LIN {X 0,Y 253.326,Z 243.578,A -85,B 0,C 180,E1 -18994.775,E2 -18994.775} C_VEL
LIN {X 0,Y 254.902,Z 232.784,A -85,B 0,C 180,E1 -18996.591,E2 -18996.591} C_VEL
LIN {X 0,Y 256.298,Z 221.635,A -85,B 0,C 180,E1 -18998.079,E2 -18998.079} C_VEL
LIN {X 0,Y 257.475,Z 209.502,A -85,B 0,C 180,E1 -18999.328,E2 -18999.328} C_VEL
LIN {X 0,Y 258.563,Z 195.963,A -85,B 0,C 180,E1 -19000.325,E2 -19000.325} C_VEL
LIN {X 0,Y 259.185,Z 183.358,A -85,B 0,C 180,E1 -19000.942,E2 -19000.942} C_VEL
LIN {X 0,Y 261.265,Z 111.221,A -85,B 0,C 180,E1 -19002.915,E2 -19002.915} C_VEL
LIN {X 0,Y 257.099,Z 99.785,A -85,B 0,C 180,E1 -19003.638,E2 -19003.638} C_VEL
LIN {X 0,Y 249.447,Z 82.487,A -85,B 0,C 180,E1 -19004.922,E2 -19004.922} C_VEL
LIN {X 0,Y 249.249,Z 81.443,A -85,B 0,C 180,E1 -19005.015,E2 -19005.015} C_VEL
LIN {X 0,Y 249.144,Z 81.454,A -85,B 0,C 180,E1 -19008.078,E2 -19008.078} C_VEL
LIN {X 0,Y 249.089,Z 81.456,A -85,B 0,C 180,E1 -19011.519,E2 -19011.519} C_VEL
LIN {X 0,Y 249.122,Z 81.453,A -85,B 0,C 180,E1 -19015.476,E2 -19015.476} C_VEL
LIN {X 0,Y 249.078,Z 81.456,A -85,B 0,C 180,E1 -19018.989,E2 -19018.989} C_VEL
LIN {X 0,Y 249.041,Z 81.457,A -85,B 0,C 180,E1 -19022.425,E2 -19022.425} C_VEL
LIN {X 0,Y 249.074,Z 81.457,A -85,B 0,C 180,E1 -19026.339,E2 -19026.339} C_VEL
LIN {X 0,Y 249.036,Z 81.46,A -85,B 0,C 180,E1 -19030.473,E2 -19030.473} C_VEL
LIN {X 0,Y 249.014,Z 81.463,A -85,B 0,C 180,E1 -19034.877,E2 -19034.877} C_VEL
LIN {X 0,Y 249.022,Z 81.466,A -85,B 0,C 180,E1 -19037.363,E2 -19037.363} C_VEL
LIN {X 0,Y 249.047,Z 81.448,A -85,B 0,C 180,E1 -19042.2,E2 -19042.2} C_VEL
LIN {X 0,Y 249.047,Z 81.441,A -85,B 0,C 180,E1 -19045.639,E2 -19045.639} C_VEL
LIN {X 0,Y 249.051,Z 81.459,A -85,B 0,C 180,E1 -19049.472,E2 -19049.472} C_VEL
LIN {X 0,Y 249.075,Z 81.456,A -85,B 0,C 180,E1 -19053.162,E2 -19053.162} C_VEL
LIN {X 0,Y 249.083,Z 81.454,A -85,B 0,C 180,E1 -19056.732,E2 -19056.732} C_VEL
LIN {X 0,Y 249.115,Z 81.455,A -85,B 0,C 180,E1 -19060.211,E2 -19060.211} C_VEL
LIN {X 0,Y 249.245,Z 81.429,A -85,B 0,C 180,E1 -19063.622,E2 -19063.622} C_VEL
LIN {X 0,Y 249.248,Z 81.436,A -85,B 0,C 180,E1 -19068.616,E2 -19068.616} C_VEL
LIN {X 0,Y 249.458,Z 81.405,A -85,B 0,C 180,E1 -19071.902,E2 -19071.902} C_VEL
LIN {X 0,Y 249.298,Z 81.429,A -85,B 0,C 180,E1 -19075.148,E2 -19075.148} C_VEL
LIN {X 0,Y 249.678,Z 81.379,A -85,B 0,C 180,E1 -19078.387,E2 -19078.387} C_VEL
LIN {X 0,Y 249.678,Z 81.379,A -85,B 0,C 180,E1 -19081.613,E2 -19081.613} C_VEL
LIN {X 0,Y 249.449,Z 81.408,A -85,B 0,C 180,E1 -19086.47,E2 -19086.47} C_VEL
LIN {X 0,Y 249.345,Z 81.425,A -85,B 0,C 180,E1 -19089.736,E2 -19089.736} C_VEL
LIN {X 0,Y 249.242,Z 81.438,A -85,B 0,C 180,E1 -19091.224,E2 -19091.224} C_VEL
LIN {X 0,Y 248.557,Z 81.529,A -85,B 0,C 180,E1 -19092.572,E2 -19092.572} C_VEL
LIN {X 0,Y 245.654,Z 81.885,A -85,B 0,C 180,E1 -19094.769,E2 -19094.769} C_VEL
LIN {X 0,Y 243.198,Z 82.185,A -85,B 0,C 180,E1 -19096.558,E2 -19096.558} C_VEL
LIN {X 0,Y 242.153,Z 82.319,A -85,B 0,C 180,E1 -19097.948,E2 -19097.948} C_VEL
LIN {X 0,Y 242.072,Z 82.328,A -85,B 0,C 180,E1 -19098.419,E2 -19098.419} C_VEL
LIN {X 0,Y 242.009,Z 82.336,A -85,B 0,C 180,E1 -19102.18,E2 -19102.18} C_VEL
LIN {X 0,Y 242.069,Z 82.328,A -85,B 0,C 180,E1 -19105.838,E2 -19105.838} C_VEL
LIN {X 0,Y 242.032,Z 82.329,A -85,B 0,C 180,E1 -19109.58,E2 -19109.58} C_VEL
LIN {X 0,Y 241.982,Z 82.341,A -85,B 0,C 180,E1 -19113.492,E2 -19113.492} C_VEL
LIN {X 0,Y 241.991,Z 82.34,A -85,B 0,C 180,E1 -19117.581,E2 -19117.581} C_VEL
LIN {X 0,Y 241.939,Z 82.348,A -85,B 0,C 180,E1 -19121.922,E2 -19121.922} C_VEL
LIN {X 0,Y 241.936,Z 82.349,A -85,B 0,C 180,E1 -19126.571,E2 -19126.571} C_VEL
LIN {X 0,Y 241.974,Z 82.346,A -85,B 0,C 180,E1 -19130.284,E2 -19130.284} C_VEL
LIN {X 0,Y 242.047,Z 82.472,A -85,B 0,C 180,E1 -19133.859,E2 -19133.859} C_VEL
LIN {X 0,Y 244.076,Z 91.796,A -85,B 0,C 180,E1 -19137.323,E2 -19137.323} C_VEL
LIN {X 0,Y 245.923,Z 100.895,A -85,B 0,C 180,E1 -19140.533,E2 -19140.533} C_VEL
LIN {X 0,Y 248.2,Z 107.794,A -85,B 0,C 180,E1 -19140.981,E2 -19140.981} C_VEL
LIN {X 0,Y 253.338,Z 152.439,A -85,B 0,C 180,E1 -19142.841,E2 -19142.841} C_VEL
LIN {X 0,Y 253.472,Z 159.178,A -85,B 0,C 180,E1 -19143.057,E2 -19143.057} C_VEL
LIN {X 0,Y 251.997,Z 209.848,A -85,B 0,C 180,E1 -19144.498,E2 -19144.498} C_VEL
LIN {X 0,Y 251.014,Z 223.134,A -85,B 0,C 180,E1 -19145.166,E2 -19145.166} C_VEL
LIN {X 0,Y 249.809,Z 235.947,A -85,B 0,C 180,E1 -19146.145,E2 -19146.145} C_VEL
LIN {X 0,Y 248.331,Z 247.285,A -85,B 0,C 180,E1 -19147.318,E2 -19147.318} C_VEL
LIN {X 0,Y 246.817,Z 257.715,A -85,B 0,C 180,E1 -19148.712,E2 -19148.712} C_VEL
LIN {X 0,Y 245.466,Z 266.328,A -85,B 0,C 180,E1 -19150.123,E2 -19150.123} C_VEL
LIN {X 0,Y 243.8,Z 276.342,A -85,B 0,C 180,E1 -19152.152,E2 -19152.152} C_VEL
LIN {X 0,Y 242.667,Z 283.898,A -85,B 0,C 180,E1 -19154.029,E2 -19154.029} C_VEL
LIN {X 0,Y 241.426,Z 292.111,A -85,B 0,C 180,E1 -19156.533,E2 -19156.533} C_VEL
LIN {X 0,Y 240.582,Z 298.702,A -85,B 0,C 180,E1 -19159.054,E2 -19159.054} C_VEL
LIN {X 0,Y 240.155,Z 303.924,A -85,B 0,C 180,E1 -19161.586,E2 -19161.586} C_VEL
LIN {X 0,Y 240.024,Z 308.554,A -85,B 0,C 180,E1 -19164.581,E2 -19164.581} C_VEL
LIN {X 0,Y 240.045,Z 310.915,A -85,B 0,C 180,E1 -19166.642,E2 -19166.642} C_VEL
LIN {X 0,Y 240.096,Z 312.31,A -85,B 0,C 180,E1 -19168.322,E2 -19168.322} C_VEL
LIN {X 0,Y 240.155,Z 313.289,A -85,B 0,C 180,E1 -19169.999,E2 -19169.999} C_VEL
LIN {X 0,Y 240.034,Z 313.858,A -85,B 0,C 180,E1 -19171.677,E2 -19171.677} C_VEL
LIN {X 0,Y 239.963,Z 314.034,A -85,B 0,C 180,E1 -19173.357,E2 -19173.357} C_VEL
LIN {X 0,Y 239.911,Z 313.751,A -85,B 0,C 180,E1 -19175.126,E2 -19175.126} C_VEL
LIN {X 0,Y 240.132,Z 312.096,A -85,B 0,C 180,E1 -19178.414,E2 -19178.414} C_VEL
LIN {X 0,Y 240.485,Z 310.677,A -85,B 0,C 180,E1 -19180.098,E2 -19180.098} C_VEL
LIN {X 0,Y 241.291,Z 307.724,A -85,B 0,C 180,E1 -19182.617,E2 -19182.617} C_VEL
LIN {X 0,Y 242.716,Z 303.775,A -85,B 0,C 180,E1 -19185.105,E2 -19185.105} C_VEL
LIN {X 0,Y 244.543,Z 298.725,A -85,B 0,C 180,E1 -19187.563,E2 -19187.563} C_VEL
LIN {X 0,Y 246.699,Z 292.425,A -85,B 0,C 180,E1 -19189.989,E2 -19189.989} C_VEL
LIN {X 0,Y 249.454,Z 284.587,A -85,B 0,C 180,E1 -19192.354,E2 -19192.354} C_VEL
LIN {X 0,Y 252.756,Z 274.849,A -85,B 0,C 180,E1 -19194.65,E2 -19194.65} C_VEL
LIN {X 0,Y 255.766,Z 264.803,A -85,B 0,C 180,E1 -19196.52,E2 -19196.52} C_VEL
LIN {X 0,Y 258.886,Z 253.45,A -85,B 0,C 180,E1 -19198.143,E2 -19198.143} C_VEL
LIN {X 0,Y 261.47,Z 242.35,A -85,B 0,C 180,E1 -19199.375,E2 -19199.375} C_VEL
LIN {X 0,Y 263.807,Z 230.005,A -85,B 0,C 180,E1 -19200.409,E2 -19200.409} C_VEL
LIN {X 0,Y 265.654,Z 216.896,A -85,B 0,C 180,E1 -19201.166,E2 -19201.166} C_VEL
LIN {X 0,Y 266.696,Z 204.407,A -85,B 0,C 180,E1 -19201.639,E2 -19201.639} C_VEL
LIN {X 0,Y 268.491,Z 159.915,A -85,B 0,C 180,E1 -19202.843,E2 -19202.843} C_VEL
LIN {X 0,Y 265.485,Z 139.44,A -85,B 0,C 180,E1 -19204.05,E2 -19204.05} C_VEL
LIN {X 0,Y 264.082,Z 132.709,A -85,B 0,C 180,E1 -19204.533,E2 -19204.533} C_VEL
LIN {X 0,Y 256.737,Z 117.087,A -85,B 0,C 180,E1 -19206.475,E2 -19206.475} C_VEL
LIN {X 0,Y 250.909,Z 106.205,A -85,B 0,C 180,E1 -19208.088,E2 -19208.088} C_VEL
LIN {X 0,Y 248.94,Z 102.739,A -85,B 0,C 180,E1 -19208.652,E2 -19208.652} C_VEL
LIN {X 0,Y 246.669,Z 98.329,A -85,B 0,C 180,E1 -19209.374,E2 -19209.374} C_VEL
LIN {X 0,Y 244.126,Z 89.558,A -85,B 0,C 180,E1 -19213.702,E2 -19213.702} C_VEL
LIN {X 0,Y 241.982,Z 82.339,A -85,B 0,C 180,E1 -19217.689,E2 -19217.689} C_VEL
LIN {X 0,Y 242.008,Z 82.331,A -85,B 0,C 180,E1 -19222.422,E2 -19222.422} C_VEL
LIN {X 0,Y 241.989,Z 82.336,A -85,B 0,C 180,E1 -19226.509,E2 -19226.509} C_VEL
LIN {X 0,Y 242.035,Z 82.333,A -85,B 0,C 180,E1 -19230.587,E2 -19230.587} C_VEL
LIN {X 0,Y 242.065,Z 82.324,A -85,B 0,C 180,E1 -19234.183,E2 -19234.183} C_VEL
LIN {X 0,Y 242.051,Z 82.322,A -85,B 0,C 180,E1 -19238.297,E2 -19238.297} C_VEL
LIN {X 0,Y 242.161,Z 82.311,A -85,B 0,C 180,E1 -19243.278,E2 -19243.278} C_VEL
LIN {X 0,Y 242.184,Z 82.306,A -85,B 0,C 180,E1 -19248.28,E2 -19248.28} C_VEL
LIN {X 0,Y 242.424,Z 82.274,A -85,B 0,C 180,E1 -19251.666,E2 -19251.666} C_VEL
LIN {X 0,Y 242.256,Z 82.309,A -85,B 0,C 180,E1 -19255.007,E2 -19255.007} C_VEL
LIN {X 0,Y 242.634,Z 82.248,A -85,B 0,C 180,E1 -19258.341,E2 -19258.341} C_VEL
LIN {X 0,Y 242.633,Z 82.252,A -85,B 0,C 180,E1 -19261.66,E2 -19261.66} C_VEL
LIN {X 0,Y 242.414,Z 82.282,A -85,B 0,C 180,E1 -19266.671,E2 -19266.671} C_VEL
LIN {X 0,Y 242.264,Z 82.307,A -85,B 0,C 180,E1 -19270.024,E2 -19270.024} C_VEL
LIN {X 0,Y 242.137,Z 82.324,A -85,B 0,C 180,E1 -19275.143,E2 -19275.143} C_VEL
LIN {X 0,Y 242.048,Z 82.327,A -85,B 0,C 180,E1 -19278.627,E2 -19278.627} C_VEL
LIN {X 0,Y 242.002,Z 82.329,A -85,B 0,C 180,E1 -19282.182,E2 -19282.182} C_VEL
LIN {X 0,Y 242.031,Z 82.327,A -85,B 0,C 180,E1 -19285.822,E2 -19285.822} C_VEL
LIN {X 0,Y 241.969,Z 82.337,A -85,B 0,C 180,E1 -19289.589,E2 -19289.589} C_VEL
LIN {X 0,Y 241.978,Z 82.342,A -85,B 0,C 180,E1 -19293.494,E2 -19293.494} C_VEL
LIN {X 0,Y 241.988,Z 82.338,A -85,B 0,C 180,E1 -19295.656,E2 -19295.656} C_VEL
LIN {X 0,Y 242.945,Z 85.113,A -85,B 0,C 180,E1 -19296.016,E2 -19296.016} C_VEL
LIN {X 0,Y 245.321,Z 87.875,A -85,B 0,C 180,E1 -19296.704,E2 -19296.704} C_VEL
LIN {X 0,Y 247.518,Z 91.21,A -85,B 0,C 180,E1 -19297.349,E2 -19297.349} C_VEL
LIN {X 0,Y 255.952,Z 103.808,A -85,B 0,C 180,E1 -19299.658,E2 -19299.658} C_VEL
LIN {X 0,Y 263.759,Z 117.045,A -85,B 0,C 180,E1 -19301.642,E2 -19301.642} C_VEL
LIN {X 0,Y 269.885,Z 129.938,A -85,B 0,C 180,E1 -19303.166,E2 -19303.166} C_VEL
LIN {X 0,Y 267.385,Z 185.069,A -85,B 0,C 180,E1 -19304.641,E2 -19304.641} C_VEL
LIN {X 0,Y 266.192,Z 198.279,A -85,B 0,C 180,E1 -19305.267,E2 -19305.267} C_VEL
LIN {X 0,Y 264.735,Z 210.283,A -85,B 0,C 180,E1 -19306.133,E2 -19306.133} C_VEL
LIN {X 0,Y 262.688,Z 221.975,A -85,B 0,C 180,E1 -19307.244,E2 -19307.244} C_VEL
LIN {X 0,Y 260.354,Z 232.814,A -85,B 0,C 180,E1 -19308.598,E2 -19308.598} C_VEL
LIN {X 0,Y 257.378,Z 244.089,A -85,B 0,C 180,E1 -19310.39,E2 -19310.39} C_VEL
LIN {X 0,Y 254.767,Z 252.802,A -85,B 0,C 180,E1 -19312.137,E2 -19312.137} C_VEL
LIN {X 0,Y 252.064,Z 260.954,A -85,B 0,C 180,E1 -19314.161,E2 -19314.161} C_VEL
LIN {X 0,Y 249.231,Z 268.801,A -85,B 0,C 180,E1 -19316.642,E2 -19316.642} C_VEL
LIN {X 0,Y 246.777,Z 275.025,A -85,B 0,C 180,E1 -19319.162,E2 -19319.162} C_VEL
LIN {X 0,Y 244.728,Z 279.883,A -85,B 0,C 180,E1 -19321.717,E2 -19321.717} C_VEL
LIN {X 0,Y 243.121,Z 283.537,A -85,B 0,C 180,E1 -19324.304,E2 -19324.304} C_VEL
LIN {X 0,Y 242.244,Z 285.369,A -85,B 0,C 180,E1 -19326.036,E2 -19326.036} C_VEL
LIN {X 0,Y 241.125,Z 287.353,A -85,B 0,C 180,E1 -19328.861,E2 -19328.861} C_VEL
LIN {X 0,Y 240.43,Z 288.166,A -85,B 0,C 180,E1 -19331.245,E2 -19331.245} C_VEL
LIN {X 0,Y 240.119,Z 288.226,A -85,B 0,C 180,E1 -19332.982,E2 -19332.982} C_VEL
LIN {X 0,Y 239.941,Z 287.748,A -85,B 0,C 180,E1 -19335.15,E2 -19335.15} C_VEL
LIN {X 0,Y 239.923,Z 285.974,A -85,B 0,C 180,E1 -19338.168,E2 -19338.168} C_VEL
LIN {X 0,Y 240.215,Z 283.416,A -85,B 0,C 180,E1 -19340.741,E2 -19340.741} C_VEL
LIN {X 0,Y 240.691,Z 279.845,A -85,B 0,C 180,E1 -19343.293,E2 -19343.293} C_VEL
LIN {X 0,Y 241.299,Z 275.174,A -85,B 0,C 180,E1 -19345.825,E2 -19345.825} C_VEL
LIN {X 0,Y 242.331,Z 268.136,A -85,B 0,C 180,E1 -19348.754,E2 -19348.754} C_VEL
LIN {X 0,Y 243.634,Z 260.515,A -85,B 0,C 180,E1 -19351.24,E2 -19351.24} C_VEL
LIN {X 0,Y 245.003,Z 252.706,A -85,B 0,C 180,E1 -19353.289,E2 -19353.289} C_VEL
LIN {X 0,Y 246.762,Z 242.095,A -85,B 0,C 180,E1 -19355.517,E2 -19355.517} C_VEL
LIN {X 0,Y 248.368,Z 231.465,A -85,B 0,C 180,E1 -19357.29,E2 -19357.29} C_VEL
LIN {X 0,Y 249.678,Z 220.807,A -85,B 0,C 180,E1 -19358.703,E2 -19358.703} C_VEL
LIN {X 0,Y 250.81,Z 209.345,A -85,B 0,C 180,E1 -19359.883,E2 -19359.883} C_VEL
LIN {X 0,Y 251.895,Z 196.367,A -85,B 0,C 180,E1 -19360.856,E2 -19360.856} C_VEL
LIN {X 0,Y 252.569,Z 183.311,A -85,B 0,C 180,E1 -19361.504,E2 -19361.504} C_VEL
LIN {X 0,Y 254.778,Z 112.933,A -85,B 0,C 180,E1 -19363.459,E2 -19363.459} C_VEL
LIN {X 0,Y 250.712,Z 101.974,A -85,B 0,C 180,E1 -19364.188,E2 -19364.188} C_VEL
LIN {X 0,Y 242.289,Z 82.759,A -85,B 0,C 180,E1 -19365.676,E2 -19365.676} C_VEL
LIN {X 0,Y 242.22,Z 82.318,A -85,B 0,C 180,E1 -19365.705,E2 -19365.705} C_VEL
LIN {X 0,Y 242.041,Z 82.337,A -85,B 0,C 180,E1 -19370.392,E2 -19370.392} C_VEL
LIN {X 0,Y 242.046,Z 82.334,A -85,B 0,C 180,E1 -19373.986,E2 -19373.986} C_VEL
LIN {X 0,Y 242.005,Z 82.332,A -85,B 0,C 180,E1 -19377.688,E2 -19377.688} C_VEL
LIN {X 0,Y 241.98,Z 82.343,A -85,B 0,C 180,E1 -19381.52,E2 -19381.52} C_VEL
LIN {X 0,Y 242.033,Z 82.331,A -85,B 0,C 180,E1 -19385.604,E2 -19385.604} C_VEL
LIN {X 0,Y 241.98,Z 82.34,A -85,B 0,C 180,E1 -19389.715,E2 -19389.715} C_VEL
LIN {X 0,Y 241.945,Z 82.342,A -85,B 0,C 180,E1 -19394.199,E2 -19394.199} C_VEL
LIN {X 0,Y 241.943,Z 82.345,A -85,B 0,C 180,E1 -19398.078,E2 -19398.078} C_VEL
LIN {X 0,Y 241.99,Z 82.325,A -85,B 0,C 180,E1 -19402.417,E2 -19402.417} C_VEL
LIN {X 0,Y 241.984,Z 82.323,A -85,B 0,C 180,E1 -19406.507,E2 -19406.507} C_VEL
LIN {X 0,Y 242.017,Z 82.337,A -85,B 0,C 180,E1 -19410.597,E2 -19410.597} C_VEL
LIN {X 0,Y 242.071,Z 82.328,A -85,B 0,C 180,E1 -19414.183,E2 -19414.183} C_VEL
LIN {X 0,Y 242.057,Z 82.332,A -85,B 0,C 180,E1 -19418.297,E2 -19418.297} C_VEL
LIN {X 0,Y 242.167,Z 82.31,A -85,B 0,C 180,E1 -19423.278,E2 -19423.278} C_VEL
LIN {X 0,Y 242.184,Z 82.318,A -85,B 0,C 180,E1 -19428.279,E2 -19428.279} C_VEL
LIN {X 0,Y 242.404,Z 82.283,A -85,B 0,C 180,E1 -19431.664,E2 -19431.664} C_VEL
LIN {X 0,Y 242.259,Z 82.305,A -85,B 0,C 180,E1 -19435.007,E2 -19435.007} C_VEL
LIN {X 0,Y 242.638,Z 82.256,A -85,B 0,C 180,E1 -19438.34,E2 -19438.34} C_VEL
LIN {X 0,Y 242.638,Z 82.256,A -85,B 0,C 180,E1 -19441.659,E2 -19441.659} C_VEL
LIN {X 0,Y 242.419,Z 82.283,A -85,B 0,C 180,E1 -19446.659,E2 -19446.659} C_VEL
LIN {X 0,Y 242.269,Z 82.305,A -85,B 0,C 180,E1 -19450.023,E2 -19450.023} C_VEL
LIN {X 0,Y 242.169,Z 82.314,A -85,B 0,C 180,E1 -19455.14,E2 -19455.14} C_VEL
LIN {X 0,Y 242.072,Z 82.328,A -85,B 0,C 180,E1 -19458.419,E2 -19458.419} C_VEL
LIN {X 0,Y 241.403,Z 82.42,A -85,B 0,C 180,E1 -19459.807,E2 -19459.807} C_VEL
LIN {X 0,Y 238.508,Z 82.78,A -85,B 0,C 180,E1 -19462.069,E2 -19462.069} C_VEL
LIN {X 0,Y 236.063,Z 83.078,A -85,B 0,C 180,E1 -19463.913,E2 -19463.913} C_VEL
LIN {X 0,Y 235.044,Z 83.204,A -85,B 0,C 180,E1 -19465.346,E2 -19465.346} C_VEL
LIN {X 0,Y 234.978,Z 83.211,A -85,B 0,C 180,E1 -19465.831,E2 -19465.831} C_VEL
LIN {X 0,Y 234.934,Z 83.213,A -85,B 0,C 180,E1 -19470.567,E2 -19470.567} C_VEL
LIN {X 0,Y 234.932,Z 83.221,A -85,B 0,C 180,E1 -19474.637,E2 -19474.637} C_VEL
LIN {X 0,Y 234.943,Z 83.217,A -85,B 0,C 180,E1 -19478.944,E2 -19478.944} C_VEL
LIN {X 0,Y 234.889,Z 83.222,A -85,B 0,C 180,E1 -19483.485,E2 -19483.485} C_VEL
LIN {X 0,Y 234.889,Z 83.227,A -85,B 0,C 180,E1 -19486.514,E2 -19486.514} C_VEL
LIN {X 0,Y 234.956,Z 83.22,A -85,B 0,C 180,E1 -19491.086,E2 -19491.086} C_VEL
LIN {X 0,Y 234.994,Z 83.241,A -85,B 0,C 180,E1 -19493.262,E2 -19493.262} C_VEL
LIN {X 0,Y 237.003,Z 92.535,A -85,B 0,C 180,E1 -19496.84,E2 -19496.84} C_VEL
LIN {X 0,Y 238.655,Z 100.654,A -85,B 0,C 180,E1 -19499.751,E2 -19499.751} C_VEL
LIN {X 0,Y 241.824,Z 109.835,A -85,B 0,C 180,E1 -19500.391,E2 -19500.391} C_VEL
LIN {X 0,Y 246.655,Z 152.06,A -85,B 0,C 180,E1 -19502.213,E2 -19502.213} C_VEL
LIN {X 0,Y 246.901,Z 159.165,A -85,B 0,C 180,E1 -19502.458,E2 -19502.458} C_VEL
LIN {X 0,Y 245.349,Z 209.737,A -85,B 0,C 180,E1 -19503.933,E2 -19503.933} C_VEL
LIN {X 0,Y 244.291,Z 223.619,A -85,B 0,C 180,E1 -19504.663,E2 -19504.663} C_VEL
LIN {X 0,Y 243.041,Z 236.191,A -85,B 0,C 180,E1 -19505.665,E2 -19505.665} C_VEL
LIN {X 0,Y 241.514,Z 247.358,A -85,B 0,C 180,E1 -19506.868,E2 -19506.868} C_VEL
LIN {X 0,Y 239.954,Z 257.708,A -85,B 0,C 180,E1 -19508.298,E2 -19508.298} C_VEL
LIN {X 0,Y 238.562,Z 266.26,A -85,B 0,C 180,E1 -19509.747,E2 -19509.747} C_VEL
LIN {X 0,Y 236.806,Z 276.349,A -85,B 0,C 180,E1 -19511.861,E2 -19511.861} C_VEL
LIN {X 0,Y 235.515,Z 284.49,A -85,B 0,C 180,E1 -19513.976,E2 -19513.976} C_VEL
LIN {X 0,Y 234.268,Z 292.53,A -85,B 0,C 180,E1 -19516.555,E2 -19516.555} C_VEL
LIN {X 0,Y 233.555,Z 297.962,A -85,B 0,C 180,E1 -19518.72,E2 -19518.72} C_VEL
LIN {X 0,Y 233.095,Z 303.268,A -85,B 0,C 180,E1 -19521.329,E2 -19521.329} C_VEL
LIN {X 0,Y 232.935,Z 307.488,A -85,B 0,C 180,E1 -19524.025,E2 -19524.025} C_VEL
LIN {X 0,Y 232.957,Z 310.378,A -85,B 0,C 180,E1 -19526.54,E2 -19526.54} C_VEL
LIN {X 0,Y 233.021,Z 311.828,A -85,B 0,C 180,E1 -19528.271,E2 -19528.271} C_VEL
LIN {X 0,Y 233.075,Z 312.834,A -85,B 0,C 180,E1 -19529.999,E2 -19529.999} C_VEL
LIN {X 0,Y 232.959,Z 313.431,A -85,B 0,C 180,E1 -19531.728,E2 -19531.728} C_VEL
LIN {X 0,Y 232.878,Z 313.637,A -85,B 0,C 180,E1 -19533.46,E2 -19533.46} C_VEL
LIN {X 0,Y 232.839,Z 313.434,A -85,B 0,C 180,E1 -19535.195,E2 -19535.195} C_VEL
LIN {X 0,Y 233.08,Z 311.809,A -85,B 0,C 180,E1 -19538.671,E2 -19538.671} C_VEL
LIN {X 0,Y 233.466,Z 310.42,A -85,B 0,C 180,E1 -19540.405,E2 -19540.405} C_VEL
LIN {X 0,Y 234.33,Z 307.529,A -85,B 0,C 180,E1 -19542.999,E2 -19542.999} C_VEL
LIN {X 0,Y 235.854,Z 303.646,A -85,B 0,C 180,E1 -19545.555,E2 -19545.555} C_VEL
LIN {X 0,Y 237.77,Z 298.666,A -85,B 0,C 180,E1 -19548.08,E2 -19548.08} C_VEL
LIN {X 0,Y 240.035,Z 292.442,A -85,B 0,C 180,E1 -19550.569,E2 -19550.569} C_VEL
LIN {X 0,Y 242.902,Z 284.737,A -85,B 0,C 180,E1 -19552.991,E2 -19552.991} C_VEL
LIN {X 0,Y 246.342,Z 275.105,A -85,B 0,C 180,E1 -19555.336,E2 -19555.336} C_VEL
LIN {X 0,Y 249.46,Z 265.208,A -85,B 0,C 180,E1 -19557.245,E2 -19557.245} C_VEL
LIN {X 0,Y 252.69,Z 254.091,A -85,B 0,C 180,E1 -19558.897,E2 -19558.897} C_VEL
LIN {X 0,Y 255.343,Z 243.237,A -85,B 0,C 180,E1 -19560.152,E2 -19560.152} C_VEL
LIN {X 0,Y 257.75,Z 231.286,A -85,B 0,C 180,E1 -19561.202,E2 -19561.202} C_VEL
LIN {X 0,Y 259.732,Z 218.262,A -85,B 0,C 180,E1 -19562.017,E2 -19562.017} C_VEL
LIN {X 0,Y 260.945,Z 205.409,A -85,B 0,C 180,E1 -19562.534,E2 -19562.534} C_VEL
LIN {X 0,Y 262.874,Z 160.81,A -85,B 0,C 180,E1 -19563.766,E2 -19563.766} C_VEL
LIN {X 0,Y 259.723,Z 139.333,A -85,B 0,C 180,E1 -19565.093,E2 -19565.093} C_VEL
LIN {X 0,Y 258.858,Z 135.778,A -85,B 0,C 180,E1 -19565.382,E2 -19565.382} C_VEL
LIN {X 0,Y 252.112,Z 121.264,A -85,B 0,C 180,E1 -19567.252,E2 -19567.252} C_VEL
LIN {X 0,Y 245.295,Z 108.243,A -85,B 0,C 180,E1 -19569.251,E2 -19569.251} C_VEL
LIN {X 0,Y 241.807,Z 102.388,A -85,B 0,C 180,E1 -19570.314,E2 -19570.314} C_VEL
LIN {X 0,Y 239.248,Z 97.728,A -85,B 0,C 180,E1 -19571.193,E2 -19571.193} C_VEL
LIN {X 0,Y 236.609,Z 88.756,A -85,B 0,C 180,E1 -19575.958,E2 -19575.958} C_VEL
LIN {X 0,Y 234.924,Z 83.215,A -85,B 0,C 180,E1 -19579.267,E2 -19579.267} C_VEL
LIN {X 0,Y 234.955,Z 83.218,A -85,B 0,C 180,E1 -19583.863,E2 -19583.863} C_VEL
LIN {X 0,Y 234.958,Z 83.219,A -85,B 0,C 180,E1 -19587.425,E2 -19587.425} C_VEL
LIN {X 0,Y 234.95,Z 83.219,A -85,B 0,C 180,E1 -19591.406,E2 -19591.406} C_VEL
LIN {X 0,Y 234.986,Z 83.215,A -85,B 0,C 180,E1 -19595.247,E2 -19595.247} C_VEL
LIN {X 0,Y 235.01,Z 83.205,A -85,B 0,C 180,E1 -19598.97,E2 -19598.97} C_VEL
LIN {X 0,Y 235.094,Z 83.189,A -85,B 0,C 180,E1 -19603.059,E2 -19603.059} C_VEL
LIN {X 0,Y 235.116,Z 83.183,A -85,B 0,C 180,E1 -19607.922,E2 -19607.922} C_VEL
LIN {X 0,Y 235.374,Z 83.154,A -85,B 0,C 180,E1 -19611.414,E2 -19611.414} C_VEL
LIN {X 0,Y 235.4,Z 83.148,A -85,B 0,C 180,E1 -19613.142,E2 -19613.142} C_VEL
LIN {X 0,Y 235.593,Z 83.124,A -85,B 0,C 180,E1 -19618.291,E2 -19618.291} C_VEL
LIN {X 0,Y 235.593,Z 83.128,A -85,B 0,C 180,E1 -19621.71,E2 -19621.71} C_VEL
LIN {X 0,Y 235.365,Z 83.157,A -85,B 0,C 180,E1 -19626.86,E2 -19626.86} C_VEL
LIN {X 0,Y 235.21,Z 83.187,A -85,B 0,C 180,E1 -19630.328,E2 -19630.328} C_VEL
LIN {X 0,Y 235.084,Z 83.202,A -85,B 0,C 180,E1 -19635.609,E2 -19635.609} C_VEL
LIN {X 0,Y 234.989,Z 83.211,A -85,B 0,C 180,E1 -19639.208,E2 -19639.208} C_VEL
LIN {X 0,Y 234.948,Z 83.212,A -85,B 0,C 180,E1 -19642.885,E2 -19642.885} C_VEL
LIN {X 0,Y 234.945,Z 83.213,A -85,B 0,C 180,E1 -19646.661,E2 -19646.661} C_VEL
LIN {X 0,Y 234.898,Z 83.224,A -85,B 0,C 180,E1 -19650.573,E2 -19650.573} C_VEL
LIN {X 0,Y 234.923,Z 83.224,A -85,B 0,C 180,E1 -19653.849,E2 -19653.849} C_VEL
LIN {X 0,Y 235.728,Z 85.726,A -85,B 0,C 180,E1 -19654.189,E2 -19654.189} C_VEL
LIN {X 0,Y 237.702,Z 88.027,A -85,B 0,C 180,E1 -19654.816,E2 -19654.816} C_VEL
LIN {X 0,Y 238.457,Z 88.997,A -85,B 0,C 180,E1 -19655.055,E2 -19655.055} C_VEL
LIN {X 0,Y 240.8,Z 92.379,A -85,B 0,C 180,E1 -19655.797,E2 -19655.797} C_VEL
LIN {X 0,Y 247.3,Z 101.831,A -85,B 0,C 180,E1 -19657.727,E2 -19657.727} C_VEL
LIN {X 0,Y 254.457,Z 113.2,A -85,B 0,C 180,E1 -19659.708,E2 -19659.708} C_VEL
LIN {X 0,Y 259.691,Z 122.45,A -85,B 0,C 180,E1 -19661.077,E2 -19661.077} C_VEL
LIN {X 0,Y 264.293,Z 132.322,A -85,B 0,C 180,E1 -19662.275,E2 -19662.275} C_VEL
LIN {X 0,Y 261.732,Z 185.483,A -85,B 0,C 180,E1 -19663.715,E2 -19663.715} C_VEL
LIN {X 0,Y 260.499,Z 198.638,A -85,B 0,C 180,E1 -19664.348,E2 -19664.348} C_VEL
LIN {X 0,Y 258.928,Z 210.934,A -85,B 0,C 180,E1 -19665.251,E2 -19665.251} C_VEL
LIN {X 0,Y 256.909,Z 221.945,A -85,B 0,C 180,E1 -19666.312,E2 -19666.312} C_VEL
LIN {X 0,Y 254.482,Z 232.889,A -85,B 0,C 180,E1 -19667.689,E2 -19667.689} C_VEL
LIN {X 0,Y 251.84,Z 242.724,A -85,B 0,C 180,E1 -19669.248,E2 -19669.248} C_VEL
LIN {X 0,Y 248.944,Z 252.044,A -85,B 0,C 180,E1 -19671.087,E2 -19671.087} C_VEL
LIN {X 0,Y 246.067,Z 260.393,A -85,B 0,C 180,E1 -19673.146,E2 -19673.146} C_VEL
LIN {X 0,Y 243.513,Z 267.245,A -85,B 0,C 180,E1 -19675.25,E2 -19675.25} C_VEL
LIN {X 0,Y 240.855,Z 273.859,A -85,B 0,C 180,E1 -19677.802,E2 -19677.802} C_VEL
LIN {X 0,Y 238.913,Z 278.315,A -85,B 0,C 180,E1 -19679.995,E2 -19679.995} C_VEL
LIN {X 0,Y 236.8,Z 282.86,A -85,B 0,C 180,E1 -19682.921,E2 -19682.921} C_VEL
LIN {X 0,Y 235.474,Z 285.508,A -85,B 0,C 180,E1 -19685.302,E2 -19685.302} C_VEL
LIN {X 0,Y 234.151,Z 287.752,A -85,B 0,C 180,E1 -19688.509,E2 -19688.509} C_VEL
LIN {X 0,Y 233.49,Z 288.491,A -85,B 0,C 180,E1 -19690.665,E2 -19690.665} C_VEL
LIN {X 0,Y 233.112,Z 288.646,A -85,B 0,C 180,E1 -19692.454,E2 -19692.454} C_VEL
LIN {X 0,Y 232.885,Z 288.139,A -85,B 0,C 180,E1 -19694.952,E2 -19694.952} C_VEL
LIN {X 0,Y 232.828,Z 286.574,A -85,B 0,C 180,E1 -19697.802,E2 -19697.802} C_VEL
LIN {X 0,Y 232.943,Z 285.032,A -85,B 0,C 180,E1 -19699.571,E2 -19699.571} C_VEL
LIN {X 0,Y 233.352,Z 281.91,A -85,B 0,C 180,E1 -19702.211,E2 -19702.211} C_VEL
LIN {X 0,Y 233.937,Z 277.73,A -85,B 0,C 180,E1 -19704.83,E2 -19704.83} C_VEL
LIN {X 0,Y 234.878,Z 271.365,A -85,B 0,C 180,E1 -19707.857,E2 -19707.857} C_VEL
LIN {X 0,Y 236.071,Z 264.435,A -85,B 0,C 180,E1 -19710.427,E2 -19710.427} C_VEL
LIN {X 0,Y 237.628,Z 255.745,A -85,B 0,C 180,E1 -19712.967,E2 -19712.967} C_VEL
LIN {X 0,Y 239.199,Z 246.836,A -85,B 0,C 180,E1 -19715.057,E2 -19715.057} C_VEL
LIN {X 0,Y 240.907,Z 236.178,A -85,B 0,C 180,E1 -19717.069,E2 -19717.069} C_VEL
LIN {X 0,Y 242.488,Z 224.76,A -85,B 0,C 180,E1 -19718.753,E2 -19718.753} C_VEL
LIN {X 0,Y 243.901,Z 212.348,A -85,B 0,C 180,E1 -19720.166,E2 -19720.166} C_VEL
LIN {X 0,Y 245.018,Z 199.734,A -85,B 0,C 180,E1 -19721.217,E2 -19721.217} C_VEL
LIN {X 0,Y 245.825,Z 186.411,A -85,B 0,C 180,E1 -19721.961,E2 -19721.961} C_VEL
LIN {X 0,Y 246.716,Z 160.059,A -85,B 0,C 180,E1 -19722.769,E2 -19722.769} C_VEL
LIN {X 0,Y 248.193,Z 114.466,A -85,B 0,C 180,E1 -19724.049,E2 -19724.049} C_VEL
LIN {X 0,Y 244.458,Z 104.522,A -85,B 0,C 180,E1 -19724.744,E2 -19724.744} C_VEL
LIN {X 0,Y 236.349,Z 86.349,A -85,B 0,C 180,E1 -19726.222,E2 -19726.222} C_VEL
LIN {X 0,Y 235.291,Z 83.998,A -85,B 0,C 180,E1 -19726.422,E2 -19726.422} C_VEL
LIN {X 0,Y 235.136,Z 83.201,A -85,B 0,C 180,E1 -19726.497,E2 -19726.497} C_VEL
LIN {X 0,Y 235.003,Z 83.211,A -85,B 0,C 180,E1 -19731.032,E2 -19731.032} C_VEL
LIN {X 0,Y 234.998,Z 83.208,A -85,B 0,C 180,E1 -19736.206,E2 -19736.206} C_VEL
LIN {X 0,Y 234.928,Z 83.221,A -85,B 0,C 180,E1 -19740.569,E2 -19740.569} C_VEL
LIN {X 0,Y 234.965,Z 83.208,A -85,B 0,C 180,E1 -19744.633,E2 -19744.633} C_VEL
LIN {X 0,Y 234.946,Z 83.218,A -85,B 0,C 180,E1 -19748.944,E2 -19748.944} C_VEL
LIN {X 0,Y 234.931,Z 83.219,A -85,B 0,C 180,E1 -19753.477,E2 -19753.477} C_VEL
LIN {X 0,Y 234.894,Z 83.221,A -85,B 0,C 180,E1 -19756.515,E2 -19756.515} C_VEL
LIN {X 0,Y 234.922,Z 83.211,A -85,B 0,C 180,E1 -19761.079,E2 -19761.079} C_VEL
LIN {X 0,Y 234.93,Z 83.193,A -85,B 0,C 180,E1 -19765.361,E2 -19765.361} C_VEL
LIN {X 0,Y 234.926,Z 83.219,A -85,B 0,C 180,E1 -19769.431,E2 -19769.431} C_VEL
LIN {X 0,Y 234.997,Z 83.209,A -85,B 0,C 180,E1 -19773.794,E2 -19773.794} C_VEL
LIN {X 0,Y 235.015,Z 83.21,A -85,B 0,C 180,E1 -19778.97,E2 -19778.97} C_VEL
LIN {X 0,Y 235.1,Z 83.19,A -85,B 0,C 180,E1 -19783.059,E2 -19783.059} C_VEL
LIN {X 0,Y 235.118,Z 83.197,A -85,B 0,C 180,E1 -19787.922,E2 -19787.922} C_VEL
LIN {X 0,Y 235.334,Z 83.163,A -85,B 0,C 180,E1 -19791.412,E2 -19791.412} C_VEL
LIN {X 0,Y 235.377,Z 83.158,A -85,B 0,C 180,E1 -19793.14,E2 -19793.14} C_VEL
LIN {X 0,Y 235.598,Z 83.133,A -85,B 0,C 180,E1 -19798.29,E2 -19798.29} C_VEL
LIN {X 0,Y 235.598,Z 83.133,A -85,B 0,C 180,E1 -19801.709,E2 -19801.709} C_VEL
LIN {X 0,Y 235.37,Z 83.162,A -85,B 0,C 180,E1 -19806.859,E2 -19806.859} C_VEL
LIN {X 0,Y 235.216,Z 83.183,A -85,B 0,C 180,E1 -19810.327,E2 -19810.327} C_VEL
LIN {X 0,Y 235.116,Z 83.191,A -85,B 0,C 180,E1 -19815.606,E2 -19815.606} C_VEL
LIN {X 0,Y 235.01,Z 83.212,A -85,B 0,C 180,E1 -19819.205,E2 -19819.205} C_VEL
LIN {X 0,Y 234.955,Z 83.218,A -85,B 0,C 180,E1 -19822.883,E2 -19822.883} C_VEL
LIN {X 0,Y 234.978,Z 83.211,A -85,B 0,C 180,E1 -19825.831,E2 -19825.831} C_VEL
LIN {X 0,Y 234.683,Z 83.252,A -85,B 0,C 180,E1 -19826.788,E2 -19826.788} C_VEL
LIN {X 0,Y 233.324,Z 83.419,A -85,B 0,C 180,E1 -19828.2,E2 -19828.2} C_VEL
LIN {X 0,Y 228.939,Z 83.963,A -85,B 0,C 180,E1 -19831.495,E2 -19831.495} C_VEL
LIN {X 0,Y 227.926,Z 84.093,A -85,B 0,C 180,E1 -19832.974,E2 -19832.974} C_VEL
LIN {X 0,Y 227.871,Z 84.097,A -85,B 0,C 180,E1 -19833.475,E2 -19833.475} C_VEL
LIN {X 0,Y 227.893,Z 84.098,A -85,B 0,C 180,E1 -19836.695,E2 -19836.695} C_VEL
LIN {X 0,Y 227.828,Z 84.104,A -85,B 0,C 180,E1 -19840.376,E2 -19840.376} C_VEL
LIN {X 0,Y 227.835,Z 84.096,A -85,B 0,C 180,E1 -19845.192,E2 -19845.192} C_VEL
LIN {X 0,Y 227.835,Z 84.107,A -85,B 0,C 180,E1 -19849.625,E2 -19849.625} C_VEL
LIN {X 0,Y 227.958,Z 84.149,A -85,B 0,C 180,E1 -19852.684,E2 -19852.684} C_VEL
LIN {X 0,Y 229.783,Z 92.531,A -85,B 0,C 180,E1 -19856.038,E2 -19856.038} C_VEL
LIN {X 0,Y 231.313,Z 99.941,A -85,B 0,C 180,E1 -19858.876,E2 -19858.876} C_VEL
LIN {X 0,Y 235.459,Z 111.484,A -85,B 0,C 180,E1 -19859.755,E2 -19859.755} C_VEL
LIN {X 0,Y 240.194,Z 154.024,A -85,B 0,C 180,E1 -19861.646,E2 -19861.646} C_VEL
LIN {X 0,Y 240.218,Z 163.938,A -85,B 0,C 180,E1 -19861.967,E2 -19861.967} C_VEL
LIN {X 0,Y 238.739,Z 209.398,A -85,B 0,C 180,E1 -19863.329,E2 -19863.329} C_VEL
LIN {X 0,Y 237.619,Z 223.29,A -85,B 0,C 180,E1 -19864.075,E2 -19864.075} C_VEL
LIN {X 0,Y 236.395,Z 235.3,A -85,B 0,C 180,E1 -19865.052,E2 -19865.052} C_VEL
LIN {X 0,Y 234.713,Z 247.409,A -85,B 0,C 180,E1 -19866.391,E2 -19866.391} C_VEL
LIN {X 0,Y 233.105,Z 257.68,A -85,B 0,C 180,E1 -19867.859,E2 -19867.859} C_VEL
LIN {X 0,Y 231.666,Z 266.171,A -85,B 0,C 180,E1 -19869.349,E2 -19869.349} C_VEL
LIN {X 0,Y 229.88,Z 276.073,A -85,B 0,C 180,E1 -19871.491,E2 -19871.491} C_VEL
LIN {X 0,Y 228.671,Z 283.56,A -85,B 0,C 180,E1 -19873.483,E2 -19873.483} C_VEL
LIN {X 0,Y 227.343,Z 291.701,A -85,B 0,C 180,E1 -19876.138,E2 -19876.138} C_VEL
LIN {X 0,Y 226.536,Z 297.203,A -85,B 0,C 180,E1 -19878.366,E2 -19878.366} C_VEL
LIN {X 0,Y 226.052,Z 302.588,A -85,B 0,C 180,E1 -19881.056,E2 -19881.056} C_VEL
LIN {X 0,Y 225.845,Z 306.756,A -85,B 0,C 180,E1 -19883.747,E2 -19883.747} C_VEL
LIN {X 0,Y 225.872,Z 309.831,A -85,B 0,C 180,E1 -19886.432,E2 -19886.432} C_VEL
LIN {X 0,Y 225.946,Z 311.339,A -85,B 0,C 180,E1 -19888.217,E2 -19888.217} C_VEL
LIN {X 0,Y 225.998,Z 312.378,A -85,B 0,C 180,E1 -19889.999,E2 -19889.999} C_VEL
LIN {X 0,Y 225.886,Z 313.003,A -85,B 0,C 180,E1 -19891.782,E2 -19891.782} C_VEL
LIN {X 0,Y 225.772,Z 313.122,A -85,B 0,C 180,E1 -19895.049,E2 -19895.049} C_VEL
LIN {X 0,Y 225.761,Z 312.495,A -85,B 0,C 180,E1 -19897.152,E2 -19897.152} C_VEL
LIN {X 0,Y 226.462,Z 310.164,A -85,B 0,C 180,E1 -19900.731,E2 -19900.731} C_VEL
LIN {X 0,Y 227.39,Z 307.334,A -85,B 0,C 180,E1 -19903.403,E2 -19903.403} C_VEL
LIN {X 0,Y 229.012,Z 303.517,A -85,B 0,C 180,E1 -19906.033,E2 -19906.033} C_VEL
LIN {X 0,Y 231.022,Z 298.606,A -85,B 0,C 180,E1 -19908.627,E2 -19908.627} C_VEL
LIN {X 0,Y 233.379,Z 292.459,A -85,B 0,C 180,E1 -19911.184,E2 -19911.184} C_VEL
LIN {X 0,Y 236.37,Z 284.865,A -85,B 0,C 180,E1 -19913.665,E2 -19913.665} C_VEL
LIN {X 0,Y 239.338,Z 277.134,A -85,B 0,C 180,E1 -19915.665,E2 -19915.665} C_VEL
LIN {X 0,Y 242.817,Z 266.683,A -85,B 0,C 180,E1 -19917.821,E2 -19917.821} C_VEL
LIN {X 0,Y 246.143,Z 256.068,A -85,B 0,C 180,E1 -19919.506,E2 -19919.506} C_VEL
LIN {X 0,Y 248.841,Z 245.844,A -85,B 0,C 180,E1 -19920.79,E2 -19920.79} C_VEL
LIN {X 0,Y 251.565,Z 233.708,A -85,B 0,C 180,E1 -19921.941,E2 -19921.941} C_VEL
LIN {X 0,Y 253.694,Z 221.022,A -85,B 0,C 180,E1 -19922.815,E2 -19922.815} C_VEL
LIN {X 0,Y 255.17,Z 207.871,A -85,B 0,C 180,E1 -19923.425,E2 -19923.425} C_VEL
LIN {X 0,Y 257.333,Z 161.889,A -85,B 0,C 180,E1 -19924.724,E2 -19924.724} C_VEL
LIN {X 0,Y 254.487,Z 141.885,A -85,B 0,C 180,E1 -19925.997,E2 -19925.997} C_VEL
LIN {X 0,Y 253.628,Z 138.6,A -85,B 0,C 180,E1 -19926.289,E2 -19926.289} C_VEL
LIN {X 0,Y 246.584,Z 123.433,A -85,B 0,C 180,E1 -19928.351,E2 -19928.351} C_VEL
LIN {X 0,Y 240.403,Z 111.802,A -85,B 0,C 180,E1 -19930.256,E2 -19930.256} C_VEL
LIN {X 0,Y 237.683,Z 107.09,A -85,B 0,C 180,E1 -19931.135,E2 -19931.135} C_VEL
LIN {X 0,Y 234.721,Z 102.179,A -85,B 0,C 180,E1 -19932.123,E2 -19932.123} C_VEL
LIN {X 0,Y 232.038,Z 97.746,A -85,B 0,C 180,E1 -19933.056,E2 -19933.056} C_VEL
LIN {X 0,Y 231.72,Z 96.962,A -85,B 0,C 180,E1 -19933.289,E2 -19933.289} C_VEL
LIN {X 0,Y 229.554,Z 89.289,A -85,B 0,C 180,E1 -19937.659,E2 -19937.659} C_VEL
LIN {X 0,Y 227.901,Z 84.097,A -85,B 0,C 180,E1 -19940.999,E2 -19940.999} C_VEL
LIN {X 0,Y 227.899,Z 84.098,A -85,B 0,C 180,E1 -19944.132,E2 -19944.132} C_VEL
LIN {X 0,Y 227.871,Z 84.094,A -85,B 0,C 180,E1 -19948.378,E2 -19948.378} C_VEL
LIN {X 0,Y 227.884,Z 84.09,A -85,B 0,C 180,E1 -19952.445,E2 -19952.445} C_VEL
LIN {X 0,Y 227.912,Z 84.087,A -85,B 0,C 180,E1 -19956.367,E2 -19956.367} C_VEL
LIN {X 0,Y 227.941,Z 84.091,A -85,B 0,C 180,E1 -19960.175,E2 -19960.175} C_VEL
LIN {X 0,Y 228.055,Z 84.074,A -85,B 0,C 180,E1 -19963.898,E2 -19963.898} C_VEL
LIN {X 0,Y 228.073,Z 84.058,A -85,B 0,C 180,E1 -19967.544,E2 -19967.544} C_VEL
LIN {X 0,Y 228.303,Z 84.037,A -85,B 0,C 180,E1 -19971.146,E2 -19971.146} C_VEL
LIN {X 0,Y 228.351,Z 84.025,A -85,B 0,C 180,E1 -19972.929,E2 -19972.929} C_VEL
LIN {X 0,Y 228.552,Z 84,A -85,B 0,C 180,E1 -19978.238,E2 -19978.238} C_VEL
LIN {X 0,Y 228.551,Z 84.004,A -85,B 0,C 180,E1 -19981.763,E2 -19981.763} C_VEL
LIN {X 0,Y 228.316,Z 84.033,A -85,B 0,C 180,E1 -19987.073,E2 -19987.073} C_VEL
LIN {X 0,Y 228.14,Z 84.068,A -85,B 0,C 180,E1 -19990.652,E2 -19990.652} C_VEL
LIN {X 0,Y 228.039,Z 84.072,A -85,B 0,C 180,E1 -19994.274,E2 -19994.274} C_VEL
LIN {X 0,Y 227.967,Z 84.076,A -85,B 0,C 180,E1 -19997.957,E2 -19997.957} C_VEL
LIN {X 0,Y 227.92,Z 84.083,A -85,B 0,C 180,E1 -20002.324,E2 -20002.324} C_VEL
LIN {X 0,Y 227.922,Z 84.087,A -85,B 0,C 180,E1 -20006.594,E2 -20006.594} C_VEL
LIN {X 0,Y 227.873,Z 84.096,A -85,B 0,C 180,E1 -20010.282,E2 -20010.282} C_VEL
LIN {X 0,Y 227.886,Z 84.222,A -85,B 0,C 180,E1 -20011.88,E2 -20011.88} C_VEL
LIN {X 0,Y 228.879,Z 86.93,A -85,B 0,C 180,E1 -20012.309,E2 -20012.309} C_VEL
LIN {X 0,Y 231.108,Z 89.191,A -85,B 0,C 180,E1 -20013.067,E2 -20013.067} C_VEL
LIN {X 0,Y 233.48,Z 92.913,A -85,B 0,C 180,E1 -20013.905,E2 -20013.905} C_VEL
LIN {X 0,Y 235.06,Z 94.836,A -85,B 0,C 180,E1 -20014.422,E2 -20014.422} C_VEL
LIN {X 0,Y 241.018,Z 103.42,A -85,B 0,C 180,E1 -20016.322,E2 -20016.322} C_VEL
LIN {X 0,Y 248.536,Z 115.131,A -85,B 0,C 180,E1 -20018.532,E2 -20018.532} C_VEL
LIN {X 0,Y 255.036,Z 126.624,A -85,B 0,C 180,E1 -20020.328,E2 -20020.328} C_VEL
LIN {X 0,Y 258.681,Z 134.436,A -85,B 0,C 180,E1 -20021.32,E2 -20021.32} C_VEL
LIN {X 0,Y 256.128,Z 186.538,A -85,B 0,C 180,E1 -20022.779,E2 -20022.779} C_VEL
LIN {X 0,Y 254.763,Z 200.139,A -85,B 0,C 180,E1 -20023.461,E2 -20023.461} C_VEL
LIN {X 0,Y 253.132,Z 212.008,A -85,B 0,C 180,E1 -20024.364,E2 -20024.364} C_VEL
LIN {X 0,Y 250.852,Z 223.703,A -85,B 0,C 180,E1 -20025.541,E2 -20025.541} C_VEL
LIN {X 0,Y 247.976,Z 235.681,A -85,B 0,C 180,E1 -20027.142,E2 -20027.142} C_VEL
LIN {X 0,Y 244.857,Z 246.34,A -85,B 0,C 180,E1 -20028.962,E2 -20028.962} C_VEL
LIN {X 0,Y 241.951,Z 254.948,A -85,B 0,C 180,E1 -20030.82,E2 -20030.82} C_VEL
LIN {X 0,Y 238.917,Z 263.086,A -85,B 0,C 180,E1 -20033.015,E2 -20033.015} C_VEL
LIN {X 0,Y 235.964,Z 270.455,A -85,B 0,C 180,E1 -20035.536,E2 -20035.536} C_VEL
LIN {X 0,Y 233.285,Z 276.507,A -85,B 0,C 180,E1 -20038.184,E2 -20038.184} C_VEL
LIN {X 0,Y 231.045,Z 281.207,A -85,B 0,C 180,E1 -20040.877,E2 -20040.877} C_VEL
LIN {X 0,Y 229.801,Z 283.646,A -85,B 0,C 180,E1 -20042.695,E2 -20042.695} C_VEL
LIN {X 0,Y 228.737,Z 285.618,A -85,B 0,C 180,E1 -20044.523,E2 -20044.523} C_VEL
LIN {X 0,Y 227.892,Z 287.143,A -85,B 0,C 180,E1 -20046.366,E2 -20046.366} C_VEL
LIN {X 0,Y 227.166,Z 288.181,A -85,B 0,C 180,E1 -20048.208,E2 -20048.208} C_VEL
LIN {X 0,Y 226.558,Z 288.809,A -85,B 0,C 180,E1 -20050.049,E2 -20050.049} C_VEL
LIN {X 0,Y 226.124,Z 289.036,A -85,B 0,C 180,E1 -20051.893,E2 -20051.893} C_VEL
LIN {X 0,Y 225.804,Z 288.523,A -85,B 0,C 180,E1 -20054.768,E2 -20054.768} C_VEL
LIN {X 0,Y 225.718,Z 287.144,A -85,B 0,C 180,E1 -20057.412,E2 -20057.412} C_VEL
LIN {X 0,Y 225.839,Z 285.697,A -85,B 0,C 180,E1 -20059.239,E2 -20059.239} C_VEL
LIN {X 0,Y 226.219,Z 282.678,A -85,B 0,C 180,E1 -20061.964,E2 -20061.964} C_VEL
LIN {X 0,Y 226.816,Z 278.611,A -85,B 0,C 180,E1 -20064.667,E2 -20064.667} C_VEL
LIN {X 0,Y 227.754,Z 272.374,A -85,B 0,C 180,E1 -20067.79,E2 -20067.79} C_VEL
LIN {X 0,Y 228.921,Z 265.587,A -85,B 0,C 180,E1 -20070.44,E2 -20070.44} C_VEL
LIN {X 0,Y 230.51,Z 257.138,A -85,B 0,C 180,E1 -20073.059,E2 -20073.059} C_VEL
LIN {X 0,Y 232.113,Z 248.428,A -85,B 0,C 180,E1 -20075.212,E2 -20075.212} C_VEL
LIN {X 0,Y 233.779,Z 238.404,A -85,B 0,C 180,E1 -20077.216,E2 -20077.216} C_VEL
LIN {X 0,Y 235.501,Z 227.069,A -85,B 0,C 180,E1 -20079.015,E2 -20079.015} C_VEL
LIN {X 0,Y 237.025,Z 215.142,A -85,B 0,C 180,E1 -20080.464,E2 -20080.464} C_VEL
LIN {X 0,Y 238.06,Z 204.09,A -85,B 0,C 180,E1 -20081.495,E2 -20081.495} C_VEL
LIN {X 0,Y 239.013,Z 190.602,A -85,B 0,C 180,E1 -20082.387,E2 -20082.387} C_VEL
LIN {X 0,Y 239.582,Z 177.103,A -85,B 0,C 180,E1 -20082.911,E2 -20082.911} C_VEL
LIN {X 0,Y 241.507,Z 115.473,A -85,B 0,C 180,E1 -20084.701,E2 -20084.701} C_VEL
LIN {X 0,Y 235.991,Z 101.723,A -85,B 0,C 180,E1 -20085.751,E2 -20085.751} C_VEL
LIN {X 0,Y 229.099,Z 87.01,A -85,B 0,C 180,E1 -20087.057,E2 -20087.057} C_VEL
LIN {X 0,Y 228.04,Z 84.083,A -85,B 0,C 180,E1 -20087.329,E2 -20087.329} C_VEL
LIN {X 0,Y 227.921,Z 84.089,A -85,B 0,C 180,E1 -20092.321,E2 -20092.321} C_VEL
LIN {X 0,Y 227.946,Z 84.084,A -85,B 0,C 180,E1 -20096.602,E2 -20096.602} C_VEL
LIN {X 0,Y 227.902,Z 84.097,A -85,B 0,C 180,E1 -20100.291,E2 -20100.291} C_VEL
LIN {X 0,Y 227.894,Z 84.085,A -85,B 0,C 180,E1 -20103.718,E2 -20103.718} C_VEL
LIN {X 0,Y 227.874,Z 84.099,A -85,B 0,C 180,E1 -20108.086,E2 -20108.086} C_VEL
LIN {X 0,Y 227.871,Z 84.099,A -85,B 0,C 180,E1 -20112.729,E2 -20112.729} C_VEL
LIN {X 0,Y 227.817,Z 84.106,A -85,B 0,C 180,E1 -20117.258,E2 -20117.258} C_VEL
LIN {X 0,Y 227.847,Z 84.087,A -85,B 0,C 180,E1 -20121.909,E2 -20121.909} C_VEL
LIN {X 0,Y 227.883,Z 84.076,A -85,B 0,C 180,E1 -20126.377,E2 -20126.377} C_VEL
LIN {X 0,Y 227.908,Z 84.093,A -85,B 0,C 180,E1 -20130.436,E2 -20130.436} C_VEL
LIN {X 0,Y 227.932,Z 84.087,A -85,B 0,C 180,E1 -20134.426,E2 -20134.426} C_VEL
LIN {X 0,Y 227.966,Z 84.086,A -85,B 0,C 180,E1 -20138.287,E2 -20138.287} C_VEL
LIN {X 0,Y 228.038,Z 84.07,A -85,B 0,C 180,E1 -20142.825,E2 -20142.825} C_VEL
LIN {X 0,Y 228.076,Z 84.073,A -85,B 0,C 180,E1 -20147.543,E2 -20147.543} C_VEL
LIN {X 0,Y 228.271,Z 84.042,A -85,B 0,C 180,E1 -20151.144,E2 -20151.144} C_VEL
LIN {X 0,Y 228.327,Z 84.036,A -85,B 0,C 180,E1 -20152.927,E2 -20152.927} C_VEL
LIN {X 0,Y 228.557,Z 84.01,A -85,B 0,C 180,E1 -20158.237,E2 -20158.237} C_VEL
LIN {X 0,Y 228.556,Z 84.01,A -85,B 0,C 180,E1 -20161.762,E2 -20161.762} C_VEL
LIN {X 0,Y 228.321,Z 84.04,A -85,B 0,C 180,E1 -20167.072,E2 -20167.072} C_VEL
LIN {X 0,Y 228.147,Z 84.063,A -85,B 0,C 180,E1 -20170.651,E2 -20170.651} C_VEL
LIN {X 0,Y 228.065,Z 84.071,A -85,B 0,C 180,E1 -20174.272,E2 -20174.272} C_VEL
LIN {X 0,Y 228.005,Z 84.082,A -85,B 0,C 180,E1 -20177.953,E2 -20177.953} C_VEL
LIN {X 0,Y 227.919,Z 84.092,A -85,B 0,C 180,E1 -20182.32,E2 -20182.32} C_VEL
LIN {X 0,Y 227.945,Z 84.09,A -85,B 0,C 180,E1 -20186.602,E2 -20186.602} C_VEL
LIN {X 0,Y 227.911,Z 84.087,A -85,B 0,C 180,E1 -20190.296,E2 -20190.296} C_VEL
LIN {X 0,Y 227.871,Z 84.097,A -85,B 0,C 180,E1 -20193.475,E2 -20193.475} C_VEL
LIN {X 0,Y 227.604,Z 84.137,A -85,B 0,C 180,E1 -20194.46,E2 -20194.46} C_VEL
LIN {X 0,Y 226.28,Z 84.304,A -85,B 0,C 180,E1 -20195.915,E2 -20195.915} C_VEL
LIN {X 0,Y 221.901,Z 84.841,A -85,B 0,C 180,E1 -20199.312,E2 -20199.312} C_VEL
LIN {X 0,Y 220.838,Z 84.977,A -85,B 0,C 180,E1 -20200.836,E2 -20200.836} C_VEL
LIN {X 0,Y 220.757,Z 84.983,A -85,B 0,C 180,E1 -20201.354,E2 -20201.354} C_VEL
LIN {X 0,Y 220.776,Z 84.977,A -85,B 0,C 180,E1 -20205.546,E2 -20205.546} C_VEL
LIN {X 0,Y 220.812,Z 84.982,A -85,B 0,C 180,E1 -20210.464,E2 -20210.464} C_VEL
LIN {X 0,Y 220.907,Z 85.127,A -85,B 0,C 180,E1 -20212.091,E2 -20212.091} C_VEL
LIN {X 0,Y 222.997,Z 94.515,A -85,B 0,C 180,E1 -20215.984,E2 -20215.984} C_VEL
LIN {X 0,Y 224.027,Z 99.782,A -85,B 0,C 180,E1 -20217.995,E2 -20217.995} C_VEL
LIN {X 0,Y 229.147,Z 113.538,A -85,B 0,C 180,E1 -20219.099,E2 -20219.099} C_VEL
LIN {X 0,Y 233.676,Z 154.697,A -85,B 0,C 180,E1 -20220.996,E2 -20220.996} C_VEL
LIN {X 0,Y 233.648,Z 165.261,A -85,B 0,C 180,E1 -20221.343,E2 -20221.343} C_VEL
LIN {X 0,Y 232.134,Z 209.456,A -85,B 0,C 180,E1 -20222.708,E2 -20222.708} C_VEL
LIN {X 0,Y 230.99,Z 222.967,A -85,B 0,C 180,E1 -20223.456,E2 -20223.456} C_VEL
LIN {X 0,Y 229.659,Z 235.508,A -85,B 0,C 180,E1 -20224.51,E2 -20224.51} C_VEL
LIN {X 0,Y 227.929,Z 247.46,A -85,B 0,C 180,E1 -20225.885,E2 -20225.885} C_VEL
LIN {X 0,Y 226.27,Z 257.652,A -85,B 0,C 180,E1 -20227.395,E2 -20227.395} C_VEL
LIN {X 0,Y 224.618,Z 267.172,A -85,B 0,C 180,E1 -20229.15,E2 -20229.15} C_VEL
LIN {X 0,Y 222.953,Z 275.829,A -85,B 0,C 180,E1 -20231.105,E2 -20231.105} C_VEL
LIN {X 0,Y 221.521,Z 284.132,A -85,B 0,C 180,E1 -20233.409,E2 -20233.409} C_VEL
LIN {X 0,Y 220.188,Z 292.079,A -85,B 0,C 180,E1 -20236.149,E2 -20236.149} C_VEL
LIN {X 0,Y 219.301,Z 298.414,A -85,B 0,C 180,E1 -20238.913,E2 -20238.913} C_VEL
LIN {X 0,Y 218.875,Z 303.444,A -85,B 0,C 180,E1 -20241.691,E2 -20241.691} C_VEL
LIN {X 0,Y 218.773,Z 307.675,A -85,B 0,C 180,E1 -20244.785,E2 -20244.785} C_VEL
LIN {X 0,Y 218.873,Z 310.832,A -85,B 0,C 180,E1 -20248.159,E2 -20248.159} C_VEL
LIN {X 0,Y 218.922,Z 311.921,A -85,B 0,C 180,E1 -20249.999,E2 -20249.999} C_VEL
LIN {X 0,Y 218.815,Z 312.575,A -85,B 0,C 180,E1 -20251.84,E2 -20251.84} C_VEL
LIN {X 0,Y 218.699,Z 312.776,A -85,B 0,C 180,E1 -20254.999,E2 -20254.999} C_VEL
LIN {X 0,Y 218.685,Z 312.179,A -85,B 0,C 180,E1 -20257.385,E2 -20257.385} C_VEL
LIN {X 0,Y 219.434,Z 309.906,A -85,B 0,C 180,E1 -20261.079,E2 -20261.079} C_VEL
LIN {X 0,Y 220.471,Z 307.14,A -85,B 0,C 180,E1 -20263.831,E2 -20263.831} C_VEL
LIN {X 0,Y 222.188,Z 303.391,A -85,B 0,C 180,E1 -20266.539,E2 -20266.539} C_VEL
LIN {X 0,Y 224.295,Z 298.554,A -85,B 0,C 180,E1 -20269.208,E2 -20269.208} C_VEL
LIN {X 0,Y 226.764,Z 292.491,A -85,B 0,C 180,E1 -20271.833,E2 -20271.833} C_VEL
LIN {X 0,Y 229.887,Z 284.988,A -85,B 0,C 180,E1 -20274.375,E2 -20274.375} C_VEL
LIN {X 0,Y 232.978,Z 277.363,A -85,B 0,C 180,E1 -20276.419,E2 -20276.419} C_VEL
LIN {X 0,Y 236.275,Z 268.157,A -85,B 0,C 180,E1 -20278.418,E2 -20278.418} C_VEL
LIN {X 0,Y 239.616,Z 257.94,A -85,B 0,C 180,E1 -20280.15,E2 -20280.15} C_VEL
LIN {X 0,Y 242.808,Z 246.645,A -85,B 0,C 180,E1 -20281.642,E2 -20281.642} C_VEL
LIN {X 0,Y 245.591,Z 234.94,A -85,B 0,C 180,E1 -20282.814,E2 -20282.814} C_VEL
LIN {X 0,Y 247.948,Z 222.151,A -85,B 0,C 180,E1 -20283.736,E2 -20283.736} C_VEL
LIN {X 0,Y 249.503,Z 209.085,A -85,B 0,C 180,E1 -20284.386,E2 -20284.386} C_VEL
LIN {X 0,Y 251.37,Z 175.927,A -85,B 0,C 180,E1 -20285.338,E2 -20285.338} C_VEL
LIN {X 0,Y 251.826,Z 162.446,A -85,B 0,C 180,E1 -20285.752,E2 -20285.752} C_VEL
LIN {X 0,Y 249.128,Z 143.415,A -85,B 0,C 180,E1 -20287.02,E2 -20287.02} C_VEL
LIN {X 0,Y 245.06,Z 133.832,A -85,B 0,C 180,E1 -20288.272,E2 -20288.272} C_VEL
LIN {X 0,Y 238.808,Z 121.181,A -85,B 0,C 180,E1 -20290.247,E2 -20290.247} C_VEL
LIN {X 0,Y 233.589,Z 111.691,A -85,B 0,C 180,E1 -20291.995,E2 -20291.995} C_VEL
LIN {X 0,Y 230.419,Z 106.507,A -85,B 0,C 180,E1 -20293.1,E2 -20293.1} C_VEL
LIN {X 0,Y 227.315,Z 101.533,A -85,B 0,C 180,E1 -20294.232,E2 -20294.232} C_VEL
LIN {X 0,Y 224.527,Z 96.883,A -85,B 0,C 180,E1 -20295.309,E2 -20295.309} C_VEL
LIN {X 0,Y 222.837,Z 91.45,A -85,B 0,C 180,E1 -20298.524,E2 -20298.524} C_VEL
LIN {X 0,Y 220.853,Z 84.967,A -85,B 0,C 180,E1 -20302.942,E2 -20302.942} C_VEL
LIN {X 0,Y 220.822,Z 84.978,A -85,B 0,C 180,E1 -20307.245,E2 -20307.245} C_VEL
LIN {X 0,Y 220.835,Z 84.977,A -85,B 0,C 180,E1 -20311.486,E2 -20311.486} C_VEL
LIN {X 0,Y 220.866,Z 84.973,A -85,B 0,C 180,E1 -20315.565,E2 -20315.565} C_VEL
LIN {X 0,Y 220.891,Z 84.97,A -85,B 0,C 180,E1 -20319.514,E2 -20319.514} C_VEL
LIN {X 0,Y 221.014,Z 84.944,A -85,B 0,C 180,E1 -20323.37,E2 -20323.37} C_VEL
LIN {X 0,Y 221.105,Z 84.939,A -85,B 0,C 180,E1 -20329.006,E2 -20329.006} C_VEL
LIN {X 0,Y 221.286,Z 84.904,A -85,B 0,C 180,E1 -20332.702,E2 -20332.702} C_VEL
LIN {X 0,Y 221.51,Z 84.877,A -85,B 0,C 180,E1 -20338.182,E2 -20338.182} C_VEL
LIN {X 0,Y 221.509,Z 84.88,A -85,B 0,C 180,E1 -20341.819,E2 -20341.819} C_VEL
LIN {X 0,Y 221.252,Z 84.911,A -85,B 0,C 180,E1 -20347.3,E2 -20347.3} C_VEL
LIN {X 0,Y 221.06,Z 84.948,A -85,B 0,C 180,E1 -20350.997,E2 -20350.997} C_VEL
LIN {X 0,Y 220.989,Z 84.948,A -85,B 0,C 180,E1 -20356.632,E2 -20356.632} C_VEL
LIN {X 0,Y 220.877,Z 84.967,A -85,B 0,C 180,E1 -20360.488,E2 -20360.488} C_VEL
LIN {X 0,Y 220.848,Z 84.972,A -85,B 0,C 180,E1 -20364.438,E2 -20364.438} C_VEL
LIN {X 0,Y 220.804,Z 84.975,A -85,B 0,C 180,E1 -20368.519,E2 -20368.519} C_VEL
LIN {X 0,Y 220.848,Z 84.967,A -85,B 0,C 180,E1 -20369.621,E2 -20369.621} C_VEL
LIN {X 0,Y 221.704,Z 87.612,A -85,B 0,C 180,E1 -20370.084,E2 -20370.084} C_VEL
LIN {X 0,Y 223.804,Z 89.931,A -85,B 0,C 180,E1 -20370.892,E2 -20370.892} C_VEL
LIN {X 0,Y 224.538,Z 90.591,A -85,B 0,C 180,E1 -20371.16,E2 -20371.16} C_VEL
LIN {X 0,Y 226.55,Z 93.786,A -85,B 0,C 180,E1 -20371.944,E2 -20371.944} C_VEL
LIN {X 0,Y 228.125,Z 95.58,A -85,B 0,C 180,E1 -20372.504,E2 -20372.504} C_VEL
LIN {X 0,Y 230.76,Z 99.258,A -85,B 0,C 180,E1 -20373.441,E2 -20373.441} C_VEL
LIN {X 0,Y 237.221,Z 108.601,A -85,B 0,C 180,E1 -20375.598,E2 -20375.598} C_VEL
LIN {X 0,Y 244.797,Z 120.642,A -85,B 0,C 180,E1 -20377.921,E2 -20377.921} C_VEL
LIN {X 0,Y 250.632,Z 131.217,A -85,B 0,C 180,E1 -20379.606,E2 -20379.606} C_VEL
LIN {X 0,Y 253.241,Z 136.934,A -85,B 0,C 180,E1 -20380.357,E2 -20380.357} C_VEL
LIN {X 0,Y 250.625,Z 186.959,A -85,B 0,C 180,E1 -20381.769,E2 -20381.769} C_VEL
LIN {X 0,Y 249.208,Z 200.525,A -85,B 0,C 180,E1 -20382.46,E2 -20382.46} C_VEL
LIN {X 0,Y 247.385,Z 213.18,A -85,B 0,C 180,E1 -20383.446,E2 -20383.446} C_VEL
LIN {X 0,Y 244.852,Z 225.399,A -85,B 0,C 180,E1 -20384.733,E2 -20384.733} C_VEL
LIN {X 0,Y 242.099,Z 236.219,A -85,B 0,C 180,E1 -20386.219,E2 -20386.219} C_VEL
LIN {X 0,Y 238.954,Z 246.504,A -85,B 0,C 180,E1 -20388.002,E2 -20388.002} C_VEL
LIN {X 0,Y 235.589,Z 256,A -85,B 0,C 180,E1 -20390.106,E2 -20390.106} C_VEL
LIN {X 0,Y 232.397,Z 264.117,A -85,B 0,C 180,E1 -20392.38,E2 -20392.38} C_VEL
LIN {X 0,Y 229.373,Z 271.297,A -85,B 0,C 180,E1 -20394.936,E2 -20394.936} C_VEL
LIN {X 0,Y 226.94,Z 276.456,A -85,B 0,C 180,E1 -20397.254,E2 -20397.254} C_VEL
LIN {X 0,Y 224.581,Z 281.16,A -85,B 0,C 180,E1 -20399.954,E2 -20399.954} C_VEL
LIN {X 0,Y 223.188,Z 283.742,A -85,B 0,C 180,E1 -20401.849,E2 -20401.849} C_VEL
LIN {X 0,Y 222.056,Z 285.732,A -85,B 0,C 180,E1 -20403.699,E2 -20403.699} C_VEL
LIN {X 0,Y 221.114,Z 287.317,A -85,B 0,C 180,E1 -20405.595,E2 -20405.595} C_VEL
LIN {X 0,Y 220.211,Z 288.557,A -85,B 0,C 180,E1 -20407.75,E2 -20407.75} C_VEL
LIN {X 0,Y 219.157,Z 289.405,A -85,B 0,C 180,E1 -20411.297,E2 -20411.297} C_VEL
LIN {X 0,Y 218.715,Z 288.906,A -85,B 0,C 180,E1 -20414.581,E2 -20414.581} C_VEL
LIN {X 0,Y 218.632,Z 287.713,A -85,B 0,C 180,E1 -20416.997,E2 -20416.997} C_VEL
LIN {X 0,Y 218.702,Z 286.327,A -85,B 0,C 180,E1 -20418.884,E2 -20418.884} C_VEL
LIN {X 0,Y 219.082,Z 283.405,A -85,B 0,C 180,E1 -20421.701,E2 -20421.701} C_VEL
LIN {X 0,Y 219.685,Z 279.448,A -85,B 0,C 180,E1 -20424.493,E2 -20424.493} C_VEL
LIN {X 0,Y 220.477,Z 274.362,A -85,B 0,C 180,E1 -20427.26,E2 -20427.26} C_VEL
LIN {X 0,Y 221.533,Z 267.978,A -85,B 0,C 180,E1 -20430.001,E2 -20430.001} C_VEL
LIN {X 0,Y 223.1,Z 259.965,A -85,B 0,C 180,E1 -20432.709,E2 -20432.709} C_VEL
LIN {X 0,Y 224.673,Z 251.804,A -85,B 0,C 180,E1 -20434.935,E2 -20434.935} C_VEL
LIN {X 0,Y 226.495,Z 241.855,A -85,B 0,C 180,E1 -20437.13,E2 -20437.13} C_VEL
LIN {X 0,Y 228.333,Z 230.63,A -85,B 0,C 180,E1 -20439.077,E2 -20439.077} C_VEL
LIN {X 0,Y 229.793,Z 219.676,A -85,B 0,C 180,E1 -20440.575,E2 -20440.575} C_VEL
LIN {X 0,Y 231.061,Z 207.596,A -85,B 0,C 180,E1 -20441.848,E2 -20441.848} C_VEL
LIN {X 0,Y 232.16,Z 195.043,A -85,B 0,C 180,E1 -20442.784,E2 -20442.784} C_VEL
LIN {X 0,Y 232.854,Z 182.087,A -85,B 0,C 180,E1 -20443.404,E2 -20443.404} C_VEL
LIN {X 0,Y 235.031,Z 116.993,A -85,B 0,C 180,E1 -20445.349,E2 -20445.349} C_VEL
LIN {X 0,Y 228.085,Z 100.4,A -85,B 0,C 180,E1 -20446.716,E2 -20446.716} C_VEL
LIN {X 0,Y 222.158,Z 88.096,A -85,B 0,C 180,E1 -20447.897,E2 -20447.897} C_VEL
LIN {X 0,Y 221.035,Z 85.383,A -85,B 0,C 180,E1 -20448.143,E2 -20448.143} C_VEL
LIN {X 0,Y 220.963,Z 84.963,A -85,B 0,C 180,E1 -20448.24,E2 -20448.24} C_VEL
LIN {X 0,Y 220.89,Z 84.964,A -85,B 0,C 180,E1 -20452.676,E2 -20452.676} C_VEL
LIN {X 0,Y 220.887,Z 84.961,A -85,B 0,C 180,E1 -20457.014,E2 -20457.014} C_VEL
LIN {X 0,Y 220.843,Z 84.975,A -85,B 0,C 180,E1 -20460.768,E2 -20460.768} C_VEL
LIN {X 0,Y 220.819,Z 84.969,A -85,B 0,C 180,E1 -20464.952,E2 -20464.952} C_VEL
LIN {X 0,Y 220.842,Z 84.975,A -85,B 0,C 180,E1 -20467.288,E2 -20467.288} C_VEL
LIN {X 0,Y 220.82,Z 84.978,A -85,B 0,C 180,E1 -20471.942,E2 -20471.942} C_VEL
LIN {X 0,Y 220.781,Z 84.978,A -85,B 0,C 180,E1 -20475.547,E2 -20475.547} C_VEL
LIN {X 0,Y 220.81,Z 84.973,A -85,B 0,C 180,E1 -20480.463,E2 -20480.463} C_VEL
LIN {X 0,Y 220.804,Z 84.946,A -85,B 0,C 180,E1 -20485.045,E2 -20485.045} C_VEL
LIN {X 0,Y 220.837,Z 84.973,A -85,B 0,C 180,E1 -20489.389,E2 -20489.389} C_VEL
LIN {X 0,Y 220.898,Z 84.965,A -85,B 0,C 180,E1 -20493.549,E2 -20493.549} C_VEL
LIN {X 0,Y 220.882,Z 84.967,A -85,B 0,C 180,E1 -20497.553,E2 -20497.553} C_VEL
LIN {X 0,Y 220.988,Z 84.95,A -85,B 0,C 180,E1 -20502.571,E2 -20502.571} C_VEL
LIN {X 0,Y 221.015,Z 84.952,A -85,B 0,C 180,E1 -20507.138,E2 -20507.138} C_VEL
LIN {X 0,Y 221.208,Z 84.922,A -85,B 0,C 180,E1 -20510.859,E2 -20510.859} C_VEL
LIN {X 0,Y 221.262,Z 84.916,A -85,B 0,C 180,E1 -20512.7,E2 -20512.7} C_VEL
LIN {X 0,Y 221.515,Z 84.887,A -85,B 0,C 180,E1 -20518.181,E2 -20518.181} C_VEL
LIN {X 0,Y 221.514,Z 84.887,A -85,B 0,C 180,E1 -20521.818,E2 -20521.818} C_VEL
LIN {X 0,Y 221.256,Z 84.917,A -85,B 0,C 180,E1 -20527.299,E2 -20527.299} C_VEL
LIN {X 0,Y 221.069,Z 84.946,A -85,B 0,C 180,E1 -20530.996,E2 -20530.996} C_VEL
LIN {X 0,Y 221.019,Z 84.947,A -85,B 0,C 180,E1 -20536.629,E2 -20536.629} C_VEL
LIN {X 0,Y 220.887,Z 84.969,A -85,B 0,C 180,E1 -20540.486,E2 -20540.486} C_VEL
LIN {X 0,Y 220.864,Z 84.972,A -85,B 0,C 180,E1 -20544.435,E2 -20544.435} C_VEL
LIN {X 0,Y 220.839,Z 84.974,A -85,B 0,C 180,E1 -20548.513,E2 -20548.513} C_VEL
LIN {X 0,Y 220.82,Z 84.978,A -85,B 0,C 180,E1 -20552.755,E2 -20552.755} C_VEL
LIN {X 0,Y 220.812,Z 84.979,A -85,B 0,C 180,E1 -20557.278,E2 -20557.278} C_VEL
LIN {X 0,Y 220.757,Z 84.983,A -85,B 0,C 180,E1 -20561.354,E2 -20561.354} C_VEL
LIN {X 0,Y 220.102,Z 85.071,A -85,B 0,C 180,E1 -20562.876,E2 -20562.876} C_VEL
LIN {X 0,Y 217.263,Z 85.431,A -85,B 0,C 180,E1 -20565.362,E2 -20565.362} C_VEL
LIN {X 0,Y 214.841,Z 85.731,A -85,B 0,C 180,E1 -20567.392,E2 -20567.392} C_VEL
LIN {X 0,Y 213.801,Z 85.855,A -85,B 0,C 180,E1 -20568.968,E2 -20568.968} C_VEL
LIN {X 0,Y 213.716,Z 85.862,A -85,B 0,C 180,E1 -20569.503,E2 -20569.503} C_VEL
LIN {X 0,Y 213.855,Z 85.953,A -85,B 0,C 180,E1 -20571.4,E2 -20571.4} C_VEL
LIN {X 0,Y 215.895,Z 95.029,A -85,B 0,C 180,E1 -20575.322,E2 -20575.322} C_VEL
LIN {X 0,Y 216.706,Z 99.157,A -85,B 0,C 180,E1 -20577.019,E2 -20577.019} C_VEL
LIN {X 0,Y 222.951,Z 115.842,A -85,B 0,C 180,E1 -20578.43,E2 -20578.43} C_VEL
LIN {X 0,Y 227.342,Z 157.577,A -85,B 0,C 180,E1 -20580.403,E2 -20580.403} C_VEL
LIN {X 0,Y 225.625,Z 208.713,A -85,B 0,C 180,E1 -20582.019,E2 -20582.019} C_VEL
LIN {X 0,Y 224.388,Z 222.606,A -85,B 0,C 180,E1 -20582.8,E2 -20582.8} C_VEL
LIN {X 0,Y 223.052,Z 234.591,A -85,B 0,C 180,E1 -20583.824,E2 -20583.824} C_VEL
LIN {X 0,Y 221.397,Z 245.891,A -85,B 0,C 180,E1 -20585.127,E2 -20585.127} C_VEL
LIN {X 0,Y 219.451,Z 257.615,A -85,B 0,C 180,E1 -20586.901,E2 -20586.901} C_VEL
LIN {X 0,Y 217.739,Z 267.078,A -85,B 0,C 180,E1 -20588.708,E2 -20588.708} C_VEL
LIN {X 0,Y 215.777,Z 276.753,A -85,B 0,C 180,E1 -20590.991,E2 -20590.991} C_VEL
LIN {X 0,Y 214.378,Z 284.693,A -85,B 0,C 180,E1 -20593.33,E2 -20593.33} C_VEL
LIN {X 0,Y 213.046,Z 292.416,A -85,B 0,C 180,E1 -20596.162,E2 -20596.162} C_VEL
LIN {X 0,Y 212.083,Z 299.537,A -85,B 0,C 180,E1 -20599.498,E2 -20599.498} C_VEL
LIN {X 0,Y 211.733,Z 304.243,A -85,B 0,C 180,E1 -20602.37,E2 -20602.37} C_VEL
LIN {X 0,Y 211.701,Z 307.342,A -85,B 0,C 180,E1 -20604.829,E2 -20604.829} C_VEL
LIN {X 0,Y 211.801,Z 310.316,A -85,B 0,C 180,E1 -20608.098,E2 -20608.098} C_VEL
LIN {X 0,Y 211.849,Z 311.462,A -85,B 0,C 180,E1 -20609.999,E2 -20609.999} C_VEL
LIN {X 0,Y 211.743,Z 312.146,A -85,B 0,C 180,E1 -20611.901,E2 -20611.901} C_VEL
LIN {X 0,Y 211.605,Z 312.437,A -85,B 0,C 180,E1 -20614.873,E2 -20614.873} C_VEL
LIN {X 0,Y 211.623,Z 311.854,A -85,B 0,C 180,E1 -20617.633,E2 -20617.633} C_VEL
LIN {X 0,Y 211.967,Z 310.953,A -85,B 0,C 180,E1 -20619.542,E2 -20619.542} C_VEL
LIN {X 0,Y 213.073,Z 307.96,A -85,B 0,C 180,E1 -20623.349,E2 -20623.349} C_VEL
LIN {X 0,Y 214.69,Z 304.609,A -85,B 0,C 180,E1 -20626.155,E2 -20626.155} C_VEL
LIN {X 0,Y 216.759,Z 300.217,A -85,B 0,C 180,E1 -20628.918,E2 -20628.918} C_VEL
LIN {X 0,Y 219.468,Z 294.155,A -85,B 0,C 180,E1 -20631.856,E2 -20631.856} C_VEL
LIN {X 0,Y 222.852,Z 286.469,A -85,B 0,C 180,E1 -20634.699,E2 -20634.699} C_VEL
LIN {X 0,Y 226.665,Z 277.588,A -85,B 0,C 180,E1 -20637.215,E2 -20637.215} C_VEL
LIN {X 0,Y 230.067,Z 268.517,A -85,B 0,C 180,E1 -20639.258,E2 -20639.258} C_VEL
LIN {X 0,Y 233.536,Z 258.523,A -85,B 0,C 180,E1 -20641.021,E2 -20641.021} C_VEL
LIN {X 0,Y 236.832,Z 247.447,A -85,B 0,C 180,E1 -20642.537,E2 -20642.537} C_VEL
LIN {X 0,Y 239.91,Z 235.059,A -85,B 0,C 180,E1 -20643.82,E2 -20643.82} C_VEL
LIN {X 0,Y 242.356,Z 222.538,A -85,B 0,C 180,E1 -20644.75,E2 -20644.75} C_VEL
LIN {X 0,Y 244.035,Z 209.136,A -85,B 0,C 180,E1 -20645.437,E2 -20645.437} C_VEL
LIN {X 0,Y 245.567,Z 183.475,A -85,B 0,C 180,E1 -20646.207,E2 -20646.207} C_VEL
LIN {X 0,Y 246.478,Z 163.807,A -85,B 0,C 180,E1 -20646.782,E2 -20646.782} C_VEL
LIN {X 0,Y 244.104,Z 146.207,A -85,B 0,C 180,E1 -20647.987,E2 -20647.987} C_VEL
LIN {X 0,Y 237.78,Z 131.967,A -85,B 0,C 180,E1 -20650.038,E2 -20650.038} C_VEL
LIN {X 0,Y 232.251,Z 121.233,A -85,B 0,C 180,E1 -20651.92,E2 -20651.92} C_VEL
LIN {X 0,Y 227.544,Z 112.804,A -85,B 0,C 180,E1 -20653.623,E2 -20653.623} C_VEL
LIN {X 0,Y 223.537,Z 106.489,A -85,B 0,C 180,E1 -20655.136,E2 -20655.136} C_VEL
LIN {X 0,Y 220.529,Z 101.565,A -85,B 0,C 180,E1 -20656.357,E2 -20656.357} C_VEL
LIN {X 0,Y 217.54,Z 97.058,A -85,B 0,C 180,E1 -20657.621,E2 -20657.621} C_VEL
LIN {X 0,Y 216.92,Z 95.731,A -85,B 0,C 180,E1 -20658.01,E2 -20658.01} C_VEL
LIN {X 0,Y 214.909,Z 89.486,A -85,B 0,C 180,E1 -20662.338,E2 -20662.338} C_VEL
LIN {X 0,Y 213.782,Z 85.847,A -85,B 0,C 180,E1 -20665.27,E2 -20665.27} C_VEL
LIN {X 0,Y 213.794,Z 85.845,A -85,B 0,C 180,E1 -20668.724,E2 -20668.724} C_VEL
LIN {X 0,Y 213.824,Z 85.84,A -85,B 0,C 180,E1 -20672.603,E2 -20672.603} C_VEL
LIN {X 0,Y 213.85,Z 85.833,A -85,B 0,C 180,E1 -20676.953,E2 -20676.953} C_VEL
LIN {X 0,Y 213.942,Z 85.821,A -85,B 0,C 180,E1 -20682.804,E2 -20682.804} C_VEL
LIN {X 0,Y 213.952,Z 85.817,A -85,B 0,C 180,E1 -20686.707,E2 -20686.707} C_VEL
LIN {X 0,Y 214.165,Z 85.804,A -85,B 0,C 180,E1 -20690.557,E2 -20690.557} C_VEL
LIN {X 0,Y 214.225,Z 85.783,A -85,B 0,C 180,E1 -20692.46,E2 -20692.46} C_VEL
LIN {X 0,Y 214.443,Z 85.756,A -85,B 0,C 180,E1 -20698.122,E2 -20698.122} C_VEL
LIN {X 0,Y 214.548,Z 85.76,A -85,B 0,C 180,E1 -20700,E2 -20700} C_VEL
LIN {X 0,Y 214.442,Z 85.76,A -85,B 0,C 180,E1 -20701.879,E2 -20701.879} C_VEL
LIN {X 0,Y 214.192,Z 85.788,A -85,B 0,C 180,E1 -20707.542,E2 -20707.542} C_VEL
LIN {X 0,Y 213.992,Z 85.825,A -85,B 0,C 180,E1 -20711.365,E2 -20711.365} C_VEL
LIN {X 0,Y 213.908,Z 85.841,A -85,B 0,C 180,E1 -20715.239,E2 -20715.239} C_VEL
LIN {X 0,Y 213.819,Z 85.847,A -85,B 0,C 180,E1 -20719.19,E2 -20719.19} C_VEL
LIN {X 0,Y 213.802,Z 85.848,A -85,B 0,C 180,E1 -20723.233,E2 -20723.233} C_VEL
LIN {X 0,Y 213.816,Z 85.849,A -85,B 0,C 180,E1 -20727.153,E2 -20727.153} C_VEL
LIN {X 0,Y 214.563,Z 88.3,A -85,B 0,C 180,E1 -20727.581,E2 -20727.581} C_VEL
LIN {X 0,Y 216.339,Z 90.494,A -85,B 0,C 180,E1 -20728.367,E2 -20728.367} C_VEL
LIN {X 0,Y 217.667,Z 91.51,A -85,B 0,C 180,E1 -20728.902,E2 -20728.902} C_VEL
LIN {X 0,Y 219.684,Z 94.805,A -85,B 0,C 180,E1 -20729.783,E2 -20729.783} C_VEL
LIN {X 0,Y 221.525,Z 96.809,A -85,B 0,C 180,E1 -20730.505,E2 -20730.505} C_VEL
LIN {X 0,Y 225.4,Z 102.235,A -85,B 0,C 180,E1 -20732.01,E2 -20732.01} C_VEL
LIN {X 0,Y 230.835,Z 109.795,A -85,B 0,C 180,E1 -20733.952,E2 -20733.952} C_VEL
LIN {X 0,Y 238.936,Z 122.486,A -85,B 0,C 180,E1 -20736.624,E2 -20736.624} C_VEL
LIN {X 0,Y 245.808,Z 134.802,A -85,B 0,C 180,E1 -20738.715,E2 -20738.715} C_VEL
LIN {X 0,Y 247.879,Z 139.315,A -85,B 0,C 180,E1 -20739.34,E2 -20739.34} C_VEL
LIN {X 0,Y 245.23,Z 187.18,A -85,B 0,C 180,E1 -20740.704,E2 -20740.704} C_VEL
LIN {X 0,Y 243.773,Z 200.705,A -85,B 0,C 180,E1 -20741.398,E2 -20741.398} C_VEL
LIN {X 0,Y 241.881,Z 213.256,A -85,B 0,C 180,E1 -20742.381,E2 -20742.381} C_VEL
LIN {X 0,Y 239.277,Z 225.451,A -85,B 0,C 180,E1 -20743.675,E2 -20743.675} C_VEL
LIN {X 0,Y 236.371,Z 236.487,A -85,B 0,C 180,E1 -20745.21,E2 -20745.21} C_VEL
LIN {X 0,Y 233.132,Z 246.664,A -85,B 0,C 180,E1 -20746.997,E2 -20746.997} C_VEL
LIN {X 0,Y 229.965,Z 255.369,A -85,B 0,C 180,E1 -20748.925,E2 -20748.925} C_VEL
LIN {X 0,Y 226.11,Z 264.696,A -85,B 0,C 180,E1 -20751.565,E2 -20751.565} C_VEL
LIN {X 0,Y 222.785,Z 272.135,A -85,B 0,C 180,E1 -20754.297,E2 -20754.297} C_VEL
LIN {X 0,Y 219.856,Z 277.969,A -85,B 0,C 180,E1 -20757.084,E2 -20757.084} C_VEL
LIN {X 0,Y 217.401,Z 282.489,A -85,B 0,C 180,E1 -20759.93,E2 -20759.93} C_VEL
LIN {X 0,Y 215.439,Z 285.849,A -85,B 0,C 180,E1 -20762.826,E2 -20762.826} C_VEL
LIN {X 0,Y 214.379,Z 287.487,A -85,B 0,C 180,E1 -20764.775,E2 -20764.775} C_VEL
LIN {X 0,Y 213.273,Z 288.957,A -85,B 0,C 180,E1 -20767.324,E2 -20767.324} C_VEL
LIN {X 0,Y 212.2,Z 289.776,A -85,B 0,C 180,E1 -20770.659,E2 -20770.659} C_VEL
LIN {X 0,Y 211.63,Z 289.287,A -85,B 0,C 180,E1 -20774.381,E2 -20774.381} C_VEL
LIN {X 0,Y 211.561,Z 288.279,A -85,B 0,C 180,E1 -20776.554,E2 -20776.554} C_VEL
LIN {X 0,Y 211.575,Z 286.944,A -85,B 0,C 180,E1 -20778.504,E2 -20778.504} C_VEL
LIN {X 0,Y 211.93,Z 284.125,A -85,B 0,C 180,E1 -20781.418,E2 -20781.418} C_VEL
LIN {X 0,Y 212.534,Z 280.274,A -85,B 0,C 180,E1 -20784.307,E2 -20784.307} C_VEL
LIN {X 0,Y 213.327,Z 275.304,A -85,B 0,C 180,E1 -20787.168,E2 -20787.168} C_VEL
LIN {X 0,Y 214.407,Z 269.066,A -85,B 0,C 180,E1 -20790.001,E2 -20790.001} C_VEL
LIN {X 0,Y 215.989,Z 261.255,A -85,B 0,C 180,E1 -20792.798,E2 -20792.798} C_VEL
LIN {X 0,Y 217.953,Z 251.48,A -85,B 0,C 180,E1 -20795.552,E2 -20795.552} C_VEL
LIN {X 0,Y 219.766,Z 241.876,A -85,B 0,C 180,E1 -20797.706,E2 -20797.706} C_VEL
LIN {X 0,Y 221.554,Z 231.311,A -85,B 0,C 180,E1 -20799.587,E2 -20799.587} C_VEL
LIN {X 0,Y 223.064,Z 220.427,A -85,B 0,C 180,E1 -20801.127,E2 -20801.127} C_VEL
LIN {X 0,Y 224.419,Z 208.43,A -85,B 0,C 180,E1 -20802.434,E2 -20802.434} C_VEL
LIN {X 0,Y 225.546,Z 196.071,A -85,B 0,C 180,E1 -20803.401,E2 -20803.401} C_VEL
LIN {X 0,Y 226.282,Z 183.346,A -85,B 0,C 180,E1 -20804.043,E2 -20804.043} C_VEL
LIN {X 0,Y 228.514,Z 118.546,A -85,B 0,C 180,E1 -20806.038,E2 -20806.038} C_VEL
LIN {X 0,Y 220.421,Z 99.501,A -85,B 0,C 180,E1 -20807.713,E2 -20807.713} C_VEL
LIN {X 0,Y 214.052,Z 86.853,A -85,B 0,C 180,E1 -20809.048,E2 -20809.048} C_VEL
LIN {X 0,Y 213.841,Z 85.845,A -85,B 0,C 180,E1 -20809.188,E2 -20809.188} C_VEL
LIN {X 0,Y 213.815,Z 85.847,A -85,B 0,C 180,E1 -20813.231,E2 -20813.231} C_VEL
LIN {X 0,Y 213.833,Z 85.839,A -85,B 0,C 180,E1 -20817.45,E2 -20817.45} C_VEL
LIN {X 0,Y 213.774,Z 85.852,A -85,B 0,C 180,E1 -20821.737,E2 -20821.737} C_VEL
LIN {X 0,Y 213.757,Z 85.857,A -85,B 0,C 180,E1 -20826.286,E2 -20826.286} C_VEL
LIN {X 0,Y 213.745,Z 85.856,A -85,B 0,C 180,E1 -20831.118,E2 -20831.118} C_VEL
LIN {X 0,Y 213.779,Z 85.852,A -85,B 0,C 180,E1 -20833.675,E2 -20833.675} C_VEL
LIN {X 0,Y 213.716,Z 85.862,A -85,B 0,C 180,E1 -20838.875,E2 -20838.875} C_VEL
LIN {X 0,Y 213.747,Z 85.823,A -85,B 0,C 180,E1 -20843.712,E2 -20843.712} C_VEL
LIN {X 0,Y 213.784,Z 85.846,A -85,B 0,C 180,E1 -20848.731,E2 -20848.731} C_VEL
LIN {X 0,Y 213.83,Z 85.85,A -85,B 0,C 180,E1 -20852.603,E2 -20852.603} C_VEL
LIN {X 0,Y 213.856,Z 85.84,A -85,B 0,C 180,E1 -20856.953,E2 -20856.953} C_VEL
LIN {X 0,Y 213.947,Z 85.825,A -85,B 0,C 180,E1 -20862.803,E2 -20862.803} C_VEL
LIN {X 0,Y 213.957,Z 85.832,A -85,B 0,C 180,E1 -20866.706,E2 -20866.706} C_VEL
LIN {X 0,Y 214.145,Z 85.802,A -85,B 0,C 180,E1 -20870.555,E2 -20870.555} C_VEL
LIN {X 0,Y 214.103,Z 85.814,A -85,B 0,C 180,E1 -20874.348,E2 -20874.348} C_VEL
LIN {X 0,Y 214.448,Z 85.767,A -85,B 0,C 180,E1 -20878.121,E2 -20878.121} C_VEL
LIN {X 0,Y 214.553,Z 85.749,A -85,B 0,C 180,E1 -20880,E2 -20880} C_VEL
LIN {X 0,Y 214.447,Z 85.768,A -85,B 0,C 180,E1 -20881.878,E2 -20881.878} C_VEL
LIN {X 0,Y 214.196,Z 85.795,A -85,B 0,C 180,E1 -20887.541,E2 -20887.541} C_VEL
LIN {X 0,Y 214.001,Z 85.829,A -85,B 0,C 180,E1 -20891.364,E2 -20891.364} C_VEL
LIN {X 0,Y 213.935,Z 85.828,A -85,B 0,C 180,E1 -20895.236,E2 -20895.236} C_VEL
LIN {X 0,Y 213.839,Z 85.85,A -85,B 0,C 180,E1 -20899.187,E2 -20899.187} C_VEL
LIN {X 0,Y 213.813,Z 85.851,A -85,B 0,C 180,E1 -20903.231,E2 -20903.231} C_VEL
LIN {X 0,Y 213.831,Z 85.847,A -85,B 0,C 180,E1 -20907.449,E2 -20907.449} C_VEL
LIN {X 0,Y 213.779,Z 85.851,A -85,B 0,C 180,E1 -20911.735,E2 -20911.735} C_VEL
LIN {X 0,Y 213.745,Z 85.861,A -85,B 0,C 180,E1 -20916.288,E2 -20916.288} C_VEL
LIN {X 0,Y 213.714,Z 85.864,A -85,B 0,C 180,E1 -20921.125,E2 -20921.125} C_VEL
LIN {X 0,Y 213.707,Z 85.857,A -85,B 0,C 180,E1 -20923.678,E2 -20923.678} C_VEL
LIN {X 0,Y 213.709,Z 85.862,A -85,B 0,C 180,E1 -20926.343,E2 -20926.343} C_VEL
LIN {X 0,Y 213.716,Z 85.862,A -85,B 0,C 180,E1 -20929.503,E2 -20929.503} C_VEL
LIN {X 0,Y 213.161,Z 86.448,A -85,B 0,C 180,E1 -20930.538,E2 -20930.538} C_VEL
LIN {X 0,Y 211.921,Z 87.892,A -85,B 0,C 180,E1 -20931.493,E2 -20931.493} C_VEL
LIN {X 0,Y 209.224,Z 92.179,A -85,B 0,C 180,E1 -20933.273,E2 -20933.273} C_VEL
LIN {X 0,Y 208.691,Z 94.917,A -85,B 0,C 180,E1 -20934.348,E2 -20934.348} C_VEL
LIN {X 0,Y 208.742,Z 95.288,A -85,B 0,C 180,E1 -20934.506,E2 -20934.506} C_VEL
LIN {X 0,Y 209.49,Z 98.911,A -85,B 0,C 180,E1 -20935.996,E2 -20935.996} C_VEL
LIN {X 0,Y 216.658,Z 117.732,A -85,B 0,C 180,E1 -20937.696,E2 -20937.696} C_VEL
LIN {X 0,Y 220.824,Z 157.594,A -85,B 0,C 180,E1 -20939.655,E2 -20939.655} C_VEL
LIN {X 0,Y 219.089,Z 208.257,A -85,B 0,C 180,E1 -20941.303,E2 -20941.303} C_VEL
LIN {X 0,Y 217.833,Z 222.198,A -85,B 0,C 180,E1 -20942.107,E2 -20942.107} C_VEL
LIN {X 0,Y 216.367,Z 234.734,A -85,B 0,C 180,E1 -20943.212,E2 -20943.212} C_VEL
LIN {X 0,Y 214.417,Z 247.5,A -85,B 0,C 180,E1 -20944.779,E2 -20944.779} C_VEL
LIN {X 0,Y 212.649,Z 257.548,A -85,B 0,C 180,E1 -20946.376,E2 -20946.376} C_VEL
LIN {X 0,Y 210.87,Z 266.956,A -85,B 0,C 180,E1 -20948.236,E2 -20948.236} C_VEL
LIN {X 0,Y 208.769,Z 276.906,A -85,B 0,C 180,E1 -20950.679,E2 -20950.679} C_VEL
LIN {X 0,Y 207.552,Z 283.753,A -85,B 0,C 180,E1 -20952.765,E2 -20952.765} C_VEL
LIN {X 0,Y 206.118,Z 291.606,A -85,B 0,C 180,E1 -20955.687,E2 -20955.687} C_VEL
LIN {X 0,Y 205.057,Z 298.807,A -85,B 0,C 180,E1 -20959.134,E2 -20959.134} C_VEL
LIN {X 0,Y 204.665,Z 303.588,A -85,B 0,C 180,E1 -20962.104,E2 -20962.104} C_VEL
LIN {X 0,Y 204.609,Z 307.073,A -85,B 0,C 180,E1 -20964.94,E2 -20964.94} C_VEL
LIN {X 0,Y 204.728,Z 309.797,A -85,B 0,C 180,E1 -20968.032,E2 -20968.032} C_VEL
LIN {X 0,Y 204.777,Z 310.987,A -85,B 0,C 180,E1 -20969.999,E2 -20969.999} C_VEL
LIN {X 0,Y 204.671,Z 311.717,A -85,B 0,C 180,E1 -20971.967,E2 -20971.967} C_VEL
LIN {X 0,Y 204.537,Z 312.076,A -85,B 0,C 180,E1 -20974.828,E2 -20974.828} C_VEL
LIN {X 0,Y 204.584,Z 311.516,A -85,B 0,C 180,E1 -20977.897,E2 -20977.897} C_VEL
LIN {X 0,Y 204.928,Z 310.671,A -85,B 0,C 180,E1 -20979.873,E2 -20979.873} C_VEL
LIN {X 0,Y 206.132,Z 307.741,A -85,B 0,C 180,E1 -20983.807,E2 -20983.807} C_VEL
LIN {X 0,Y 207.859,Z 304.456,A -85,B 0,C 180,E1 -20986.701,E2 -20986.701} C_VEL
LIN {X 0,Y 210.043,Z 300.134,A -85,B 0,C 180,E1 -20989.547,E2 -20989.547} C_VEL
LIN {X 0,Y 212.973,Z 293.941,A -85,B 0,C 180,E1 -20992.663,E2 -20992.663} C_VEL
LIN {X 0,Y 216.424,Z 286.592,A -85,B 0,C 180,E1 -20995.484,E2 -20995.484} C_VEL
LIN {X 0,Y 220.396,Z 277.819,A -85,B 0,C 180,E1 -20998.056,E2 -20998.056} C_VEL
LIN {X 0,Y 223.906,Z 268.878,A -85,B 0,C 180,E1 -21000.146,E2 -21000.146} C_VEL
LIN {X 0,Y 227.492,Z 259.07,A -85,B 0,C 180,E1 -21001.94,E2 -21001.94} C_VEL
LIN {X 0,Y 230.892,Z 248.288,A -85,B 0,C 180,E1 -21003.483,E2 -21003.483} C_VEL
LIN {X 0,Y 234.083,Z 236.219,A -85,B 0,C 180,E1 -21004.781,E2 -21004.781} C_VEL
LIN {X 0,Y 236.755,Z 223.624,A -85,B 0,C 180,E1 -21005.761,E2 -21005.761} C_VEL
LIN {X 0,Y 238.556,Z 210.334,A -85,B 0,C 180,E1 -21006.492,E2 -21006.492} C_VEL
LIN {X 0,Y 239.83,Z 192.303,A -85,B 0,C 180,E1 -21007.072,E2 -21007.072} C_VEL
LIN {X 0,Y 241.176,Z 164.607,A -85,B 0,C 180,E1 -21007.893,E2 -21007.893} C_VEL
LIN {X 0,Y 239.097,Z 149.074,A -85,B 0,C 180,E1 -21009.004,E2 -21009.004} C_VEL
LIN {X 0,Y 233.183,Z 135.745,A -85,B 0,C 180,E1 -21011.025,E2 -21011.025} C_VEL
LIN {X 0,Y 228.189,Z 125.799,A -85,B 0,C 180,E1 -21012.824,E2 -21012.824} C_VEL
LIN {X 0,Y 223.14,Z 116.867,A -85,B 0,C 180,E1 -21014.739,E2 -21014.739} C_VEL
LIN {X 0,Y 219.996,Z 111.641,A -85,B 0,C 180,E1 -21016.006,E2 -21016.006} C_VEL
LIN {X 0,Y 216.789,Z 106.446,A -85,B 0,C 180,E1 -21017.371,E2 -21017.371} C_VEL
LIN {X 0,Y 213.316,Z 101.032,A -85,B 0,C 180,E1 -21018.939,E2 -21018.939} C_VEL
LIN {X 0,Y 210.146,Z 96.488,A -85,B 0,C 180,E1 -21020.45,E2 -21020.45} C_VEL
LIN {X 0,Y 209.478,Z 95.163,A -85,B 0,C 180,E1 -21020.819,E2 -21020.819} C_VEL
LIN {X 0,Y 207.751,Z 89.92,A -85,B 0,C 180,E1 -21024.894,E2 -21024.894} C_VEL
LIN {X 0,Y 206.723,Z 86.734,A -85,B 0,C 180,E1 -21027.711,E2 -21027.711} C_VEL
LIN {X 0,Y 206.764,Z 86.722,A -85,B 0,C 180,E1 -21032.096,E2 -21032.096} C_VEL
LIN {X 0,Y 206.783,Z 86.716,A -85,B 0,C 180,E1 -21036.584,E2 -21036.584} C_VEL
LIN {X 0,Y 206.871,Z 86.7,A -85,B 0,C 180,E1 -21042.197,E2 -21042.197} C_VEL
LIN {X 0,Y 206.895,Z 86.699,A -85,B 0,C 180,E1 -21046.245,E2 -21046.245} C_VEL
LIN {X 0,Y 207.103,Z 86.686,A -85,B 0,C 180,E1 -21050.232,E2 -21050.232} C_VEL
LIN {X 0,Y 207.165,Z 86.662,A -85,B 0,C 180,E1 -21052.201,E2 -21052.201} C_VEL
LIN {X 0,Y 207.38,Z 86.635,A -85,B 0,C 180,E1 -21058.058,E2 -21058.058} C_VEL
LIN {X 0,Y 207.513,Z 86.636,A -85,B 0,C 180,E1 -21060,E2 -21060} C_VEL
LIN {X 0,Y 207.379,Z 86.638,A -85,B 0,C 180,E1 -21061.943,E2 -21061.943} C_VEL
LIN {X 0,Y 207.135,Z 86.666,A -85,B 0,C 180,E1 -21067.801,E2 -21067.801} C_VEL
LIN {X 0,Y 206.915,Z 86.701,A -85,B 0,C 180,E1 -21071.759,E2 -21071.759} C_VEL
LIN {X 0,Y 206.842,Z 86.719,A -85,B 0,C 180,E1 -21075.773,E2 -21075.773} C_VEL
LIN {X 0,Y 206.855,Z 86.705,A -85,B 0,C 180,E1 -21077.955,E2 -21077.955} C_VEL
LIN {X 0,Y 206.745,Z 86.729,A -85,B 0,C 180,E1 -21083.392,E2 -21083.392} C_VEL
LIN {X 0,Y 206.741,Z 86.843,A -85,B 0,C 180,E1 -21084.276,E2 -21084.276} C_VEL
LIN {X 0,Y 207.524,Z 89.238,A -85,B 0,C 180,E1 -21084.778,E2 -21084.778} C_VEL
LIN {X 0,Y 209.432,Z 91.434,A -85,B 0,C 180,E1 -21085.732,E2 -21085.732} C_VEL
LIN {X 0,Y 210.822,Z 92.391,A -85,B 0,C 180,E1 -21086.361,E2 -21086.361} C_VEL
LIN {X 0,Y 212.701,Z 95.641,A -85,B 0,C 180,E1 -21087.297,E2 -21087.297} C_VEL
LIN {X 0,Y 214.904,Z 97.897,A -85,B 0,C 180,E1 -21088.259,E2 -21088.259} C_VEL
LIN {X 0,Y 217.447,Z 101.461,A -85,B 0,C 180,E1 -21089.369,E2 -21089.369} C_VEL
LIN {X 0,Y 218.669,Z 102.979,A -85,B 0,C 180,E1 -21089.874,E2 -21089.874} C_VEL
LIN {X 0,Y 225.233,Z 112.216,A -85,B 0,C 180,E1 -21092.45,E2 -21092.45} C_VEL
LIN {X 0,Y 231.738,Z 122.078,A -85,B 0,C 180,E1 -21094.763,E2 -21094.763} C_VEL
LIN {X 0,Y 238.994,Z 134.567,A -85,B 0,C 180,E1 -21097.148,E2 -21097.148} C_VEL
LIN {X 0,Y 242.502,Z 141.617,A -85,B 0,C 180,E1 -21098.254,E2 -21098.254} C_VEL
LIN {X 0,Y 239.871,Z 188.175,A -85,B 0,C 180,E1 -21099.625,E2 -21099.625} C_VEL
LIN {X 0,Y 238.298,Z 202.019,A -85,B 0,C 180,E1 -21100.363,E2 -21100.363} C_VEL
LIN {X 0,Y 236.405,Z 213.862,A -85,B 0,C 180,E1 -21101.318,E2 -21101.318} C_VEL
LIN {X 0,Y 233.788,Z 225.538,A -85,B 0,C 180,E1 -21102.567,E2 -21102.567} C_VEL
LIN {X 0,Y 230.61,Z 237.178,A -85,B 0,C 180,E1 -21104.213,E2 -21104.213} C_VEL
LIN {X 0,Y 227.015,Z 247.907,A -85,B 0,C 180,E1 -21106.157,E2 -21106.157} C_VEL
LIN {X 0,Y 222.995,Z 258.118,A -85,B 0,C 180,E1 -21108.56,E2 -21108.56} C_VEL
LIN {X 0,Y 219.71,Z 265.643,A -85,B 0,C 180,E1 -21110.821,E2 -21110.821} C_VEL
LIN {X 0,Y 216.232,Z 272.948,A -85,B 0,C 180,E1 -21113.619,E2 -21113.619} C_VEL
LIN {X 0,Y 213.679,Z 277.841,A -85,B 0,C 180,E1 -21116.005,E2 -21116.005} C_VEL
LIN {X 0,Y 211.003,Z 282.494,A -85,B 0,C 180,E1 -21118.919,E2 -21118.919} C_VEL
LIN {X 0,Y 208.851,Z 285.966,A -85,B 0,C 180,E1 -21121.894,E2 -21121.894} C_VEL
LIN {X 0,Y 207.696,Z 287.657,A -85,B 0,C 180,E1 -21123.904,E2 -21123.904} C_VEL
LIN {X 0,Y 206.361,Z 289.353,A -85,B 0,C 180,E1 -21126.86,E2 -21126.86} C_VEL
LIN {X 0,Y 205.265,Z 290.148,A -85,B 0,C 180,E1 -21129.978,E2 -21129.978} C_VEL
LIN {X 0,Y 204.815,Z 290.123,A -85,B 0,C 180,E1 -21132.012,E2 -21132.012} C_VEL
LIN {X 0,Y 204.579,Z 289.675,A -85,B 0,C 180,E1 -21134.135,E2 -21134.135} C_VEL
LIN {X 0,Y 204.462,Z 288.847,A -85,B 0,C 180,E1 -21136.078,E2 -21136.078} C_VEL
LIN {X 0,Y 204.459,Z 287.56,A -85,B 0,C 180,E1 -21138.099,E2 -21138.099} C_VEL
LIN {X 0,Y 204.806,Z 284.839,A -85,B 0,C 180,E1 -21141.118,E2 -21141.118} C_VEL
LIN {X 0,Y 205.391,Z 281.096,A -85,B 0,C 180,E1 -21144.109,E2 -21144.109} C_VEL
LIN {X 0,Y 206.18,Z 276.24,A -85,B 0,C 180,E1 -21147.07,E2 -21147.07} C_VEL
LIN {X 0,Y 207.271,Z 270.127,A -85,B 0,C 180,E1 -21150.001,E2 -21150.001} C_VEL
LIN {X 0,Y 208.852,Z 262.516,A -85,B 0,C 180,E1 -21152.894,E2 -21152.894} C_VEL
LIN {X 0,Y 210.505,Z 254.724,A -85,B 0,C 180,E1 -21155.269,E2 -21155.269} C_VEL
LIN {X 0,Y 212.386,Z 245.215,A -85,B 0,C 180,E1 -21157.607,E2 -21157.607} C_VEL
LIN {X 0,Y 214.382,Z 234.646,A -85,B 0,C 180,E1 -21159.673,E2 -21159.673} C_VEL
LIN {X 0,Y 216.109,Z 222.933,A -85,B 0,C 180,E1 -21161.49,E2 -21161.49} C_VEL
LIN {X 0,Y 217.534,Z 211.518,A -85,B 0,C 180,E1 -21162.834,E2 -21162.834} C_VEL
LIN {X 0,Y 218.846,Z 198.632,A -85,B 0,C 180,E1 -21163.938,E2 -21163.938} C_VEL
LIN {X 0,Y 219.618,Z 186.286,A -85,B 0,C 180,E1 -21164.656,E2 -21164.656} C_VEL
LIN {X 0,Y 222.055,Z 120.2,A -85,B 0,C 180,E1 -21166.761,E2 -21166.761} C_VEL
LIN {X 0,Y 213.765,Z 100.957,A -85,B 0,C 180,E1 -21168.557,E2 -21168.557} C_VEL
LIN {X 0,Y 207.813,Z 89.662,A -85,B 0,C 180,E1 -21169.85,E2 -21169.85} C_VEL
LIN {X 0,Y 206.776,Z 86.728,A -85,B 0,C 180,E1 -21170.129,E2 -21170.129} C_VEL
LIN {X 0,Y 206.752,Z 86.73,A -85,B 0,C 180,E1 -21174.074,E2 -21174.074} C_VEL
LIN {X 0,Y 206.741,Z 86.725,A -85,B 0,C 180,E1 -21178.42,E2 -21178.42} C_VEL
LIN {X 0,Y 206.71,Z 86.724,A -85,B 0,C 180,E1 -21182.956,E2 -21182.956} C_VEL
LIN {X 0,Y 206.726,Z 86.725,A -85,B 0,C 180,E1 -21185.32,E2 -21185.32} C_VEL
LIN {X 0,Y 206.683,Z 86.735,A -85,B 0,C 180,E1 -21190.247,E2 -21190.247} C_VEL
LIN {X 0,Y 206.682,Z 86.734,A -85,B 0,C 180,E1 -21194.431,E2 -21194.431} C_VEL
LIN {X 0,Y 206.665,Z 86.735,A -85,B 0,C 180,E1 -21199.749,E2 -21199.749} C_VEL
LIN {X 0,Y 206.703,Z 86.697,A -85,B 0,C 180,E1 -21204.689,E2 -21204.689} C_VEL
LIN {X 0,Y 206.711,Z 86.732,A -85,B 0,C 180,E1 -21209.336,E2 -21209.336} C_VEL
LIN {X 0,Y 206.736,Z 86.729,A -85,B 0,C 180,E1 -21213.772,E2 -21213.772} C_VEL
LIN {X 0,Y 206.762,Z 86.726,A -85,B 0,C 180,E1 -21218.043,E2 -21218.043} C_VEL
LIN {X 0,Y 206.877,Z 86.709,A -85,B 0,C 180,E1 -21222.196,E2 -21222.196} C_VEL
LIN {X 0,Y 206.899,Z 86.71,A -85,B 0,C 180,E1 -21226.244,E2 -21226.244} C_VEL
LIN {X 0,Y 207.103,Z 86.681,A -85,B 0,C 180,E1 -21230.231,E2 -21230.231} C_VEL
LIN {X 0,Y 207.064,Z 86.688,A -85,B 0,C 180,E1 -21234.155,E2 -21234.155} C_VEL
LIN {X 0,Y 207.384,Z 86.647,A -85,B 0,C 180,E1 -21238.057,E2 -21238.057} C_VEL
LIN {X 0,Y 207.518,Z 86.625,A -85,B 0,C 180,E1 -21240,E2 -21240} C_VEL
LIN {X 0,Y 207.384,Z 86.647,A -85,B 0,C 180,E1 -21241.942,E2 -21241.942} C_VEL
LIN {X 0,Y 207.139,Z 86.673,A -85,B 0,C 180,E1 -21247.8,E2 -21247.8} C_VEL
LIN {X 0,Y 206.926,Z 86.71,A -85,B 0,C 180,E1 -21251.758,E2 -21251.758} C_VEL
LIN {X 0,Y 206.868,Z 86.708,A -85,B 0,C 180,E1 -21255.77,E2 -21255.77} C_VEL
LIN {X 0,Y 206.781,Z 86.726,A -85,B 0,C 180,E1 -21259.869,E2 -21259.869} C_VEL
LIN {X 0,Y 206.749,Z 86.729,A -85,B 0,C 180,E1 -21264.074,E2 -21264.074} C_VEL
LIN {X 0,Y 206.746,Z 86.73,A -85,B 0,C 180,E1 -21268.418,E2 -21268.418} C_VEL
LIN {X 0,Y 206.704,Z 86.737,A -85,B 0,C 180,E1 -21272.956,E2 -21272.956} C_VEL
LIN {X 0,Y 206.682,Z 86.739,A -85,B 0,C 180,E1 -21277.739,E2 -21277.739} C_VEL
LIN {X 0,Y 206.643,Z 86.744,A -85,B 0,C 180,E1 -21281.562,E2 -21281.562} C_VEL
LIN {X 0,Y 206.636,Z 86.737,A -85,B 0,C 180,E1 -21285.581,E2 -21285.581} C_VEL
LIN {X 0,Y 206.724,Z 86.795,A -85,B 0,C 180,E1 -21290.654,E2 -21290.654} C_VEL
LIN {X 0,Y 208.742,Z 95.288,A -85,B 0,C 180,E1 -21294.506,E2 -21294.506} C_VEL
LIN {X 0,Y 209.219,Z 97.834,A -85,B 0,C 180,E1 -21295.282,E2 -21295.282} C_VEL
LIN {X 0,Y 209.884,Z 101.946,A -85,B 0,C 180,E1 -21295.964,E2 -21295.964} C_VEL
LIN {X 0,Y 210.417,Z 106.604,A -85,B 0,C 180,E1 -21296.398,E2 -21296.398} C_VEL
LIN {X 0,Y 211.069,Z 125.271,A -85,B 0,C 180,E1 -21297.226,E2 -21297.226} C_VEL
LIN {X 0,Y 214.389,Z 159.473,A -85,B 0,C 180,E1 -21298.936,E2 -21298.936} C_VEL
LIN {X 0,Y 212.581,Z 207.819,A -85,B 0,C 180,E1 -21300.542,E2 -21300.542} C_VEL
LIN {X 0,Y 211.399,Z 221.027,A -85,B 0,C 180,E1 -21301.315,E2 -21301.315} C_VEL
LIN {X 0,Y 209.876,Z 233.791,A -85,B 0,C 180,E1 -21302.449,E2 -21302.449} C_VEL
LIN {X 0,Y 207.946,Z 245.898,A -85,B 0,C 180,E1 -21303.936,E2 -21303.936} C_VEL
LIN {X 0,Y 206.123,Z 256.174,A -85,B 0,C 180,E1 -21305.58,E2 -21305.58} C_VEL
LIN {X 0,Y 204.186,Z 265.74,A -85,B 0,C 180,E1 -21307.485,E2 -21307.485} C_VEL
LIN {X 0,Y 202.353,Z 274.624,A -85,B 0,C 180,E1 -21309.676,E2 -21309.676} C_VEL
LIN {X 0,Y 200.753,Z 282.8,A -85,B 0,C 180,E1 -21312.162,E2 -21312.162} C_VEL
LIN {X 0,Y 199.215,Z 290.792,A -85,B 0,C 180,E1 -21315.18,E2 -21315.18} C_VEL
LIN {X 0,Y 198.283,Z 296.196,A -85,B 0,C 180,E1 -21317.721,E2 -21317.721} C_VEL
LIN {X 0,Y 197.709,Z 301.471,A -85,B 0,C 180,E1 -21320.795,E2 -21320.795} C_VEL
LIN {X 0,Y 197.514,Z 305.542,A -85,B 0,C 180,E1 -21323.871,E2 -21323.871} C_VEL
LIN {X 0,Y 197.521,Z 307.628,A -85,B 0,C 180,E1 -21325.919,E2 -21325.919} C_VEL
LIN {X 0,Y 197.633,Z 309.274,A -85,B 0,C 180,E1 -21327.961,E2 -21327.961} C_VEL
LIN {X 0,Y 197.707,Z 310.497,A -85,B 0,C 180,E1 -21329.999,E2 -21329.999} C_VEL
LIN {X 0,Y 197.6,Z 311.286,A -85,B 0,C 180,E1 -21332.038,E2 -21332.038} C_VEL
LIN {X 0,Y 197.461,Z 311.665,A -85,B 0,C 180,E1 -21334.749,E2 -21334.749} C_VEL
LIN {X 0,Y 197.536,Z 311.174,A -85,B 0,C 180,E1 -21338.181,E2 -21338.181} C_VEL
LIN {X 0,Y 197.908,Z 310.377,A -85,B 0,C 180,E1 -21340.227,E2 -21340.227} C_VEL
LIN {X 0,Y 199.208,Z 307.522,A -85,B 0,C 180,E1 -21344.297,E2 -21344.297} C_VEL
LIN {X 0,Y 201.049,Z 304.304,A -85,B 0,C 180,E1 -21347.285,E2 -21347.285} C_VEL
LIN {X 0,Y 203.358,Z 300.055,A -85,B 0,C 180,E1 -21350.217,E2 -21350.217} C_VEL
LIN {X 0,Y 206.558,Z 293.648,A -85,B 0,C 180,E1 -21353.563,E2 -21353.563} C_VEL
LIN {X 0,Y 210.048,Z 286.713,A -85,B 0,C 180,E1 -21356.316,E2 -21356.316} C_VEL
LIN {X 0,Y 214.16,Z 278.069,A -85,B 0,C 180,E1 -21358.949,E2 -21358.949} C_VEL
LIN {X 0,Y 217.815,Z 269.255,A -85,B 0,C 180,E1 -21361.08,E2 -21361.08} C_VEL
LIN {X 0,Y 221.976,Z 258.429,A -85,B 0,C 180,E1 -21363.103,E2 -21363.103} C_VEL
LIN {X 0,Y 225.515,Z 247.559,A -85,B 0,C 180,E1 -21364.662,E2 -21364.662} C_VEL
LIN {X 0,Y 228.83,Z 235.401,A -85,B 0,C 180,E1 -21365.97,E2 -21365.97} C_VEL
LIN {X 0,Y 231.514,Z 222.692,A -85,B 0,C 180,E1 -21366.972,E2 -21366.972} C_VEL
LIN {X 0,Y 233.395,Z 209.401,A -85,B 0,C 180,E1 -21367.682,E2 -21367.682} C_VEL
LIN {X 0,Y 234.705,Z 190.665,A -85,B 0,C 180,E1 -21368.288,E2 -21368.288} C_VEL
LIN {X 0,Y 235.983,Z 165.756,A -85,B 0,C 180,E1 -21369.036,E2 -21369.036} C_VEL
LIN {X 0,Y 234.246,Z 152.17,A -85,B 0,C 180,E1 -21370.036,E2 -21370.036} C_VEL
LIN {X 0,Y 228.83,Z 139.82,A -85,B 0,C 180,E1 -21371.994,E2 -21371.994} C_VEL
LIN {X 0,Y 224.117,Z 130.259,A -85,B 0,C 180,E1 -21373.785,E2 -21373.785} C_VEL
LIN {X 0,Y 219.38,Z 121.674,A -85,B 0,C 180,E1 -21375.686,E2 -21375.686} C_VEL
LIN {X 0,Y 213.833,Z 112.299,A -85,B 0,C 180,E1 -21378.103,E2 -21378.103} C_VEL
LIN {X 0,Y 210.133,Z 106.477,A -85,B 0,C 180,E1 -21379.85,E2 -21379.85} C_VEL
LIN {X 0,Y 207.034,Z 101.826,A -85,B 0,C 180,E1 -21381.412,E2 -21381.412} C_VEL
LIN {X 0,Y 205.255,Z 99.523,A -85,B 0,C 180,E1 -21382.34,E2 -21382.34} C_VEL
LIN {X 0,Y 202.094,Z 94.788,A -85,B 0,C 180,E1 -21384.144,E2 -21384.144} C_VEL
LIN {X 0,Y 201.904,Z 94.312,A -85,B 0,C 180,E1 -21384.335,E2 -21384.335} C_VEL
LIN {X 0,Y 199.961,Z 88.848,A -85,B 0,C 180,E1 -21389.361,E2 -21389.361} C_VEL
LIN {X 0,Y 199.672,Z 87.608,A -85,B 0,C 180,E1 -21390.645,E2 -21390.645} C_VEL
LIN {X 0,Y 199.671,Z 87.611,A -85,B 0,C 180,E1 -21395.016,E2 -21395.016} C_VEL
LIN {X 0,Y 199.698,Z 87.606,A -85,B 0,C 180,E1 -21399.395,E2 -21399.395} C_VEL
LIN {X 0,Y 199.803,Z 87.587,A -85,B 0,C 180,E1 -21403.657,E2 -21403.657} C_VEL
LIN {X 0,Y 200.034,Z 87.569,A -85,B 0,C 180,E1 -21409.653,E2 -21409.653} C_VEL
LIN {X 0,Y 200.109,Z 87.541,A -85,B 0,C 180,E1 -21411.925,E2 -21411.925} C_VEL
LIN {X 0,Y 200.319,Z 87.514,A -85,B 0,C 180,E1 -21417.99,E2 -21417.99} C_VEL
LIN {X 0,Y 200.477,Z 87.513,A -85,B 0,C 180,E1 -21420,E2 -21420} C_VEL
LIN {X 0,Y 200.022,Z 87.556,A -85,B 0,C 180,E1 -21424.03,E2 -21424.03} C_VEL
LIN {X 0,Y 200.084,Z 87.544,A -85,B 0,C 180,E1 -21428.077,E2 -21428.077} C_VEL
LIN {X 0,Y 199.865,Z 87.576,A -85,B 0,C 180,E1 -21432.181,E2 -21432.181} C_VEL
LIN {X 0,Y 199.786,Z 87.59,A -85,B 0,C 180,E1 -21436.346,E2 -21436.346} C_VEL
LIN {X 0,Y 199.682,Z 87.603,A -85,B 0,C 180,E1 -21440.81,E2 -21440.81} C_VEL
LIN {X 0,Y 200.545,Z 90.197,A -85,B 0,C 180,E1 -21441.523,E2 -21441.523} C_VEL
LIN {X 0,Y 202.451,Z 92.395,A -85,B 0,C 180,E1 -21442.645,E2 -21442.645} C_VEL
LIN {X 0,Y 204.025,Z 93.452,A -85,B 0,C 180,E1 -21443.471,E2 -21443.471} C_VEL
LIN {X 0,Y 205.864,Z 96.584,A -85,B 0,C 180,E1 -21444.52,E2 -21444.52} C_VEL
LIN {X 0,Y 208.224,Z 98.9,A -85,B 0,C 180,E1 -21445.691,E2 -21445.691} C_VEL
LIN {X 0,Y 210.555,Z 102.269,A -85,B 0,C 180,E1 -21446.85,E2 -21446.85} C_VEL
LIN {X 0,Y 212.229,Z 104.263,A -85,B 0,C 180,E1 -21447.621,E2 -21447.621} C_VEL
LIN {X 0,Y 216.093,Z 109.499,A -85,B 0,C 180,E1 -21449.333,E2 -21449.333} C_VEL
LIN {X 0,Y 222.026,Z 117.972,A -85,B 0,C 180,E1 -21451.753,E2 -21451.753} C_VEL
LIN {X 0,Y 228.189,Z 127.563,A -85,B 0,C 180,E1 -21454.042,E2 -21454.042} C_VEL
LIN {X 0,Y 234.556,Z 138.685,A -85,B 0,C 180,E1 -21456.238,E2 -21456.238} C_VEL
LIN {X 0,Y 237.301,Z 144.106,A -85,B 0,C 180,E1 -21457.147,E2 -21457.147} C_VEL
LIN {X 0,Y 234.692,Z 188.013,A -85,B 0,C 180,E1 -21458.442,E2 -21458.442} C_VEL
LIN {X 0,Y 233.144,Z 201.385,A -85,B 0,C 180,E1 -21459.145,E2 -21459.145} C_VEL
LIN {X 0,Y 231.119,Z 213.802,A -85,B 0,C 180,E1 -21460.139,E2 -21460.139} C_VEL
LIN {X 0,Y 228.405,Z 225.63,A -85,B 0,C 180,E1 -21461.409,E2 -21461.409} C_VEL
LIN {X 0,Y 224.975,Z 237.666,A -85,B 0,C 180,E1 -21463.131,E2 -21463.131} C_VEL
LIN {X 0,Y 221.336,Z 248.112,A -85,B 0,C 180,E1 -21465.051,E2 -21465.051} C_VEL
LIN {X 0,Y 217.528,Z 257.517,A -85,B 0,C 180,E1 -21467.276,E2 -21467.276} C_VEL
LIN {X 0,Y 213.354,Z 266.601,A -85,B 0,C 180,E1 -21470.035,E2 -21470.035} C_VEL
LIN {X 0,Y 209.705,Z 273.759,A -85,B 0,C 180,E1 -21472.898,E2 -21472.898} C_VEL
LIN {X 0,Y 206.553,Z 279.408,A -85,B 0,C 180,E1 -21475.847,E2 -21475.847} C_VEL
LIN {X 0,Y 203.819,Z 283.771,A -85,B 0,C 180,E1 -21478.855,E2 -21478.855} C_VEL
LIN {X 0,Y 202.319,Z 286.054,A -85,B 0,C 180,E1 -21480.902,E2 -21480.902} C_VEL
LIN {X 0,Y 201.064,Z 287.829,A -85,B 0,C 180,E1 -21482.974,E2 -21482.974} C_VEL
LIN {X 0,Y 199.432,Z 289.758,A -85,B 0,C 180,E1 -21486.384,E2 -21486.384} C_VEL
LIN {X 0,Y 198.361,Z 290.519,A -85,B 0,C 180,E1 -21489.25,E2 -21489.25} C_VEL
LIN {X 0,Y 197.834,Z 290.544,A -85,B 0,C 180,E1 -21491.355,E2 -21491.355} C_VEL
LIN {X 0,Y 197.509,Z 290.057,A -85,B 0,C 180,E1 -21493.896,E2 -21493.896} C_VEL
LIN {X 0,Y 197.346,Z 288.176,A -85,B 0,C 180,E1 -21497.663,E2 -21497.663} C_VEL
LIN {X 0,Y 197.643,Z 285.557,A -85,B 0,C 180,E1 -21500.793,E2 -21500.793} C_VEL
LIN {X 0,Y 198.227,Z 281.919,A -85,B 0,C 180,E1 -21503.895,E2 -21503.895} C_VEL
LIN {X 0,Y 199.036,Z 277.176,A -85,B 0,C 180,E1 -21506.965,E2 -21506.965} C_VEL
LIN {X 0,Y 200.375,Z 270.062,A -85,B 0,C 180,E1 -21510.503,E2 -21510.503} C_VEL
LIN {X 0,Y 202.064,Z 262.327,A -85,B 0,C 180,E1 -21513.49,E2 -21513.49} C_VEL
LIN {X 0,Y 204.175,Z 252.612,A -85,B 0,C 180,E1 -21516.424,E2 -21516.424} C_VEL
LIN {X 0,Y 206.278,Z 242.386,A -85,B 0,C 180,E1 -21518.863,E2 -21518.863} C_VEL
LIN {X 0,Y 208.261,Z 231.244,A -85,B 0,C 180,E1 -21520.943,E2 -21520.943} C_VEL
LIN {X 0,Y 209.938,Z 220.155,A -85,B 0,C 180,E1 -21522.569,E2 -21522.569} C_VEL
LIN {X 0,Y 211.421,Z 207.844,A -85,B 0,C 180,E1 -21523.946,E2 -21523.946} C_VEL
LIN {X 0,Y 212.619,Z 194.726,A -85,B 0,C 180,E1 -21524.966,E2 -21524.966} C_VEL
LIN {X 0,Y 213.381,Z 181.839,A -85,B 0,C 180,E1 -21525.596,E2 -21525.596} C_VEL
LIN {X 0,Y 215.605,Z 121.941,A -85,B 0,C 180,E1 -21527.526,E2 -21527.526} C_VEL
LIN {X 0,Y 208.174,Z 104.629,A -85,B 0,C 180,E1 -21529.213,E2 -21529.213} C_VEL
LIN {X 0,Y 200.743,Z 90.505,A -85,B 0,C 180,E1 -21530.923,E2 -21530.923} C_VEL
LIN {X 0,Y 199.699,Z 87.608,A -85,B 0,C 180,E1 -21531.213,E2 -21531.213} C_VEL
LIN {X 0,Y 199.669,Z 87.614,A -85,B 0,C 180,E1 -21534.986,E2 -21534.986} C_VEL
LIN {X 0,Y 199.669,Z 87.612,A -85,B 0,C 180,E1 -21539.524,E2 -21539.524} C_VEL
LIN {X 0,Y 199.662,Z 87.606,A -85,B 0,C 180,E1 -21542.349,E2 -21542.349} C_VEL
LIN {X 0,Y 199.645,Z 87.615,A -85,B 0,C 180,E1 -21546.759,E2 -21546.759} C_VEL
LIN {X 0,Y 199.645,Z 87.613,A -85,B 0,C 180,E1 -21549.32,E2 -21549.32} C_VEL
LIN {X 0,Y 199.624,Z 87.617,A -85,B 0,C 180,E1 -21552.325,E2 -21552.325} C_VEL
LIN {X 0,Y 199.6,Z 87.614,A -85,B 0,C 180,E1 -21555.233,E2 -21555.233} C_VEL
LIN {X 0,Y 199.585,Z 87.621,A -85,B 0,C 180,E1 -21558.005,E2 -21558.005} C_VEL
LIN {X 0,Y 199.614,Z 87.607,A -85,B 0,C 180,E1 -21560.767,E2 -21560.767} C_VEL
LIN {X 0,Y 199.615,Z 87.583,A -85,B 0,C 180,E1 -21565.713,E2 -21565.713} C_VEL
LIN {X 0,Y 199.697,Z 87.597,A -85,B 0,C 180,E1 -21568.136,E2 -21568.136} C_VEL
LIN {X 0,Y 199.69,Z 87.61,A -85,B 0,C 180,E1 -21572.771,E2 -21572.771} C_VEL
LIN {X 0,Y 199.742,Z 87.6,A -85,B 0,C 180,E1 -21577.229,E2 -21577.229} C_VEL
LIN {X 0,Y 199.8,Z 87.594,A -85,B 0,C 180,E1 -21581.757,E2 -21581.757} C_VEL
LIN {X 0,Y 199.839,Z 87.586,A -85,B 0,C 180,E1 -21585.748,E2 -21585.748} C_VEL
LIN {X 0,Y 200.026,Z 87.565,A -85,B 0,C 180,E1 -21589.881,E2 -21589.881} C_VEL
LIN {X 0,Y 200.026,Z 87.563,A -85,B 0,C 180,E1 -21593.949,E2 -21593.949} C_VEL
LIN {X 0,Y 200.324,Z 87.527,A -85,B 0,C 180,E1 -21597.989,E2 -21597.989} C_VEL
LIN {X 0,Y 200.482,Z 87.5,A -85,B 0,C 180,E1 -21600,E2 -21600} C_VEL
LIN {X 0,Y 200.028,Z 87.568,A -85,B 0,C 180,E1 -21604.029,E2 -21604.029} C_VEL
LIN {X 0,Y 200.088,Z 87.55,A -85,B 0,C 180,E1 -21608.076,E2 -21608.076} C_VEL
LIN {X 0,Y 199.876,Z 87.586,A -85,B 0,C 180,E1 -21612.179,E2 -21612.179} C_VEL
LIN {X 0,Y 199.806,Z 87.588,A -85,B 0,C 180,E1 -21616.343,E2 -21616.343} C_VEL
LIN {X 0,Y 199.693,Z 87.61,A -85,B 0,C 180,E1 -21620.606,E2 -21620.606} C_VEL
LIN {X 0,Y 199.667,Z 87.611,A -85,B 0,C 180,E1 -21624.985,E2 -21624.985} C_VEL
LIN {X 0,Y 199.677,Z 87.603,A -85,B 0,C 180,E1 -21629.522,E2 -21629.522} C_VEL
LIN {X 0,Y 199.68,Z 87.608,A -85,B 0,C 180,E1 -21632.358,E2 -21632.358} C_VEL
LIN {X 0,Y 199.625,Z 87.619,A -85,B 0,C 180,E1 -21636.762,E2 -21636.762} C_VEL
LIN {X 0,Y 199.61,Z 87.618,A -85,B 0,C 180,E1 -21639.327,E2 -21639.327} C_VEL
LIN {X 0,Y 199.576,Z 87.624,A -85,B 0,C 180,E1 -21642.31,E2 -21642.31} C_VEL
LIN {X 0,Y 199.582,Z 87.612,A -85,B 0,C 180,E1 -21645.228,E2 -21645.228} C_VEL
LIN {X 0,Y 199.686,Z 87.819,A -85,B 0,C 180,E1 -21649.949,E2 -21649.949} C_VEL
LIN {X 0,Y 201.57,Z 95.62,A -85,B 0,C 180,E1 -21653.648,E2 -21653.648} C_VEL
LIN {X 0,Y 202.202,Z 98.513,A -85,B 0,C 180,E1 -21654.872,E2 -21654.872} C_VEL
LIN {X 0,Y 210.184,Z 119.105,A -85,B 0,C 180,E1 -21656.869,E2 -21656.869} C_VEL
LIN {X 0,Y 211.044,Z 125.073,A -85,B 0,C 180,E1 -21657.215,E2 -21657.215} C_VEL
LIN {X 0,Y 211.069,Z 125.271,A -85,B 0,C 180,E1 -21657.226,E2 -21657.226} C_VEL
LIN {X 0,Y 211.229,Z 129.172,A -85,B 0,C 180,E1 -21657.395,E2 -21657.395} C_VEL
LIN {X 0,Y 210.148,Z 137.036,A -85,B 0,C 180,E1 -21657.545,E2 -21657.545} C_VEL
LIN {X 0,Y 207.546,Z 150.728,A -85,B 0,C 180,E1 -21657.711,E2 -21657.711} C_VEL
LIN {X 0,Y 207.717,Z 156.561,A -85,B 0,C 180,E1 -21657.957,E2 -21657.957} C_VEL
LIN {X 0,Y 207.905,Z 162.897,A -85,B 0,C 180,E1 -21658.224,E2 -21658.224} C_VEL
LIN {X 0,Y 206.117,Z 207.363,A -85,B 0,C 180,E1 -21659.734,E2 -21659.734} C_VEL
LIN {X 0,Y 204.911,Z 220.605,A -85,B 0,C 180,E1 -21660.53,E2 -21660.53} C_VEL
LIN {X 0,Y 203.426,Z 232.819,A -85,B 0,C 180,E1 -21661.637,E2 -21661.637} C_VEL
LIN {X 0,Y 201.592,Z 244.304,A -85,B 0,C 180,E1 -21663.049,E2 -21663.049} C_VEL
LIN {X 0,Y 199.367,Z 256.107,A -85,B 0,C 180,E1 -21664.974,E2 -21664.974} C_VEL
LIN {X 0,Y 197.353,Z 265.617,A -85,B 0,C 180,E1 -21666.937,E2 -21666.937} C_VEL
LIN {X 0,Y 195.463,Z 274.464,A -85,B 0,C 180,E1 -21669.203,E2 -21669.203} C_VEL
LIN {X 0,Y 193.613,Z 283.347,A -85,B 0,C 180,E1 -21672.028,E2 -21672.028} C_VEL
LIN {X 0,Y 192.069,Z 291.113,A -85,B 0,C 180,E1 -21675.158,E2 -21675.158} C_VEL
LIN {X 0,Y 191.038,Z 297.341,A -85,B 0,C 180,E1 -21678.326,E2 -21678.326} C_VEL
LIN {X 0,Y 190.545,Z 302.272,A -85,B 0,C 180,E1 -21681.515,E2 -21681.515} C_VEL
LIN {X 0,Y 190.459,Z 306.417,A -85,B 0,C 180,E1 -21685.075,E2 -21685.075} C_VEL
LIN {X 0,Y 190.541,Z 308.751,A -85,B 0,C 180,E1 -21687.885,E2 -21687.885} C_VEL
LIN {X 0,Y 190.638,Z 310.007,A -85,B 0,C 180,E1 -21689.999,E2 -21689.999} C_VEL
LIN {X 0,Y 190.508,Z 310.838,A -85,B 0,C 180,E1 -21692.113,E2 -21692.113} C_VEL
LIN {X 0,Y 190.398,Z 311.255,A -85,B 0,C 180,E1 -21694.71,E2 -21694.71} C_VEL
LIN {X 0,Y 190.488,Z 310.832,A -85,B 0,C 180,E1 -21698.486,E2 -21698.486} C_VEL
LIN {X 0,Y 191.484,Z 308.904,A -85,B 0,C 180,E1 -21702.721,E2 -21702.721} C_VEL
LIN {X 0,Y 192.302,Z 307.307,A -85,B 0,C 180,E1 -21704.822,E2 -21704.822} C_VEL
LIN {X 0,Y 194.26,Z 304.16,A -85,B 0,C 180,E1 -21707.909,E2 -21707.909} C_VEL
LIN {X 0,Y 196.7,Z 299.984,A -85,B 0,C 180,E1 -21710.933,E2 -21710.933} C_VEL
LIN {X 0,Y 200.062,Z 293.656,A -85,B 0,C 180,E1 -21714.377,E2 -21714.377} C_VEL
LIN {X 0,Y 203.703,Z 286.809,A -85,B 0,C 180,E1 -21717.202,E2 -21717.202} C_VEL
LIN {X 0,Y 207.972,Z 278.32,A -85,B 0,C 180,E1 -21719.896,E2 -21719.896} C_VEL
LIN {X 0,Y 211.792,Z 269.631,A -85,B 0,C 180,E1 -21722.068,E2 -21722.068} C_VEL
LIN {X 0,Y 216.082,Z 258.96,A -85,B 0,C 180,E1 -21724.128,E2 -21724.128} C_VEL
LIN {X 0,Y 219.731,Z 248.373,A -85,B 0,C 180,E1 -21725.712,E2 -21725.712} C_VEL
LIN {X 0,Y 223.147,Z 236.568,A -85,B 0,C 180,E1 -21727.037,E2 -21727.037} C_VEL
LIN {X 0,Y 225.97,Z 224.322,A -85,B 0,C 180,E1 -21728.038,E2 -21728.038} C_VEL
LIN {X 0,Y 228.039,Z 211.113,A -85,B 0,C 180,E1 -21728.815,E2 -21728.815} C_VEL
LIN {X 0,Y 229.188,Z 197.565,A -85,B 0,C 180,E1 -21729.309,E2 -21729.309} C_VEL
LIN {X 0,Y 230.932,Z 167.188,A -85,B 0,C 180,E1 -21730.208,E2 -21730.208} C_VEL
LIN {X 0,Y 229.441,Z 155.273,A -85,B 0,C 180,E1 -21731.126,E2 -21731.126} C_VEL
LIN {X 0,Y 224.464,Z 143.766,A -85,B 0,C 180,E1 -21733.031,E2 -21733.031} C_VEL
LIN {X 0,Y 220.085,Z 134.608,A -85,B 0,C 180,E1 -21734.795,E2 -21734.795} C_VEL
LIN {X 0,Y 215.572,Z 126.324,A -85,B 0,C 180,E1 -21736.713,E2 -21736.713} C_VEL
LIN {X 0,Y 210.365,Z 117.382,A -85,B 0,C 180,E1 -21739.111,E2 -21739.111} C_VEL
LIN {X 0,Y 207.046,Z 112.018,A -85,B 0,C 180,E1 -21740.765,E2 -21740.765} C_VEL
LIN {X 0,Y 203.173,Z 106.133,A -85,B 0,C 180,E1 -21742.85,E2 -21742.85} C_VEL
LIN {X 0,Y 199.595,Z 100.851,A -85,B 0,C 180,E1 -21744.964,E2 -21744.964} C_VEL
LIN {X 0,Y 195.191,Z 95.18,A -85,B 0,C 180,E1 -21747.845,E2 -21747.845} C_VEL
LIN {X 0,Y 194.241,Z 93.369,A -85,B 0,C 180,E1 -21748.66,E2 -21748.66} C_VEL
LIN {X 0,Y 193.208,Z 90.451,A -85,B 0,C 180,E1 -21751.779,E2 -21751.779} C_VEL
LIN {X 0,Y 192.597,Z 88.484,A -85,B 0,C 180,E1 -21754.277,E2 -21754.277} C_VEL
LIN {X 0,Y 192.704,Z 88.471,A -85,B 0,C 180,E1 -21756.349,E2 -21756.349} C_VEL
LIN {X 0,Y 192.73,Z 88.463,A -85,B 0,C 180,E1 -21761.458,E2 -21761.458} C_VEL
LIN {X 0,Y 192.763,Z 88.47,A -85,B 0,C 180,E1 -21765.214,E2 -21765.214} C_VEL
LIN {X 0,Y 192.979,Z 88.447,A -85,B 0,C 180,E1 -21769.509,E2 -21769.509} C_VEL
LIN {X 0,Y 193.059,Z 88.42,A -85,B 0,C 180,E1 -21771.628,E2 -21771.628} C_VEL
LIN {X 0,Y 193.261,Z 88.393,A -85,B 0,C 180,E1 -21777.916,E2 -21777.916} C_VEL
LIN {X 0,Y 193.441,Z 88.389,A -85,B 0,C 180,E1 -21780,E2 -21780} C_VEL
LIN {X 0,Y 192.968,Z 88.435,A -85,B 0,C 180,E1 -21784.178,E2 -21784.178} C_VEL
LIN {X 0,Y 193.032,Z 88.423,A -85,B 0,C 180,E1 -21788.375,E2 -21788.375} C_VEL
LIN {X 0,Y 192.792,Z 88.454,A -85,B 0,C 180,E1 -21792.635,E2 -21792.635} C_VEL
LIN {X 0,Y 192.74,Z 88.588,A -85,B 0,C 180,E1 -21796.824,E2 -21796.824} C_VEL
LIN {X 0,Y 193.519,Z 90.947,A -85,B 0,C 180,E1 -21797.544,E2 -21797.544} C_VEL
LIN {X 0,Y 195.742,Z 93.476,A -85,B 0,C 180,E1 -21799.125,E2 -21799.125} C_VEL
LIN {X 0,Y 197.235,Z 94.4,A -85,B 0,C 180,E1 -21800.058,E2 -21800.058} C_VEL
LIN {X 0,Y 199.045,Z 97.556,A -85,B 0,C 180,E1 -21801.286,E2 -21801.286} C_VEL
LIN {X 0,Y 201.642,Z 100.018,A -85,B 0,C 180,E1 -21802.784,E2 -21802.784} C_VEL
LIN {X 0,Y 203.986,Z 103.382,A -85,B 0,C 180,E1 -21804.12,E2 -21804.12} C_VEL
LIN {X 0,Y 205.729,Z 105.305,A -85,B 0,C 180,E1 -21805.026,E2 -21805.026} C_VEL
LIN {X 0,Y 208.552,Z 109.036,A -85,B 0,C 180,E1 -21806.453,E2 -21806.453} C_VEL
LIN {X 0,Y 213.747,Z 116.226,A -85,B 0,C 180,E1 -21808.869,E2 -21808.869} C_VEL
LIN {X 0,Y 220.332,Z 125.937,A -85,B 0,C 180,E1 -21811.623,E2 -21811.623} C_VEL
LIN {X 0,Y 226.845,Z 136.741,A -85,B 0,C 180,E1 -21814.096,E2 -21814.096} C_VEL
LIN {X 0,Y 232.191,Z 146.661,A -85,B 0,C 180,E1 -21815.987,E2 -21815.987} C_VEL
LIN {X 0,Y 229.548,Z 188.772,A -85,B 0,C 180,E1 -21817.248,E2 -21817.248} C_VEL
LIN {X 0,Y 227.863,Z 202.59,A -85,B 0,C 180,E1 -21817.999,E2 -21817.999} C_VEL
LIN {X 0,Y 225.656,Z 215.191,A -85,B 0,C 180,E1 -21819.044,E2 -21819.044} C_VEL
LIN {X 0,Y 222.656,Z 227.366,A -85,B 0,C 180,E1 -21820.405,E2 -21820.405} C_VEL
LIN {X 0,Y 219.16,Z 239.015,A -85,B 0,C 180,E1 -21822.136,E2 -21822.136} C_VEL
LIN {X 0,Y 215.331,Z 249.328,A -85,B 0,C 180,E1 -21824.108,E2 -21824.108} C_VEL
LIN {X 0,Y 211.296,Z 258.76,A -85,B 0,C 180,E1 -21826.423,E2 -21826.423} C_VEL
LIN {X 0,Y 207.734,Z 266.166,A -85,B 0,C 180,E1 -21828.723,E2 -21828.723} C_VEL
LIN {X 0,Y 203.823,Z 273.533,A -85,B 0,C 180,E1 -21831.637,E2 -21831.637} C_VEL
LIN {X 0,Y 200.445,Z 279.309,A -85,B 0,C 180,E1 -21834.654,E2 -21834.654} C_VEL
LIN {X 0,Y 197.512,Z 283.788,A -85,B 0,C 180,E1 -21837.742,E2 -21837.742} C_VEL
LIN {X 0,Y 195.857,Z 286.126,A -85,B 0,C 180,E1 -21839.844,E2 -21839.844} C_VEL
LIN {X 0,Y 194.466,Z 288,A -85,B 0,C 180,E1 -21841.978,E2 -21841.978} C_VEL
LIN {X 0,Y 192.531,Z 290.162,A -85,B 0,C 180,E1 -21845.866,E2 -21845.866} C_VEL
LIN {X 0,Y 191.51,Z 290.865,A -85,B 0,C 180,E1 -21848.472,E2 -21848.472} C_VEL
LIN {X 0,Y 190.89,Z 290.964,A -85,B 0,C 180,E1 -21850.65,E2 -21850.65} C_VEL
LIN {X 0,Y 190.449,Z 290.44,A -85,B 0,C 180,E1 -21853.633,E2 -21853.633} C_VEL
LIN {X 0,Y 190.251,Z 288.786,A -85,B 0,C 180,E1 -21857.195,E2 -21857.195} C_VEL
LIN {X 0,Y 190.492,Z 286.263,A -85,B 0,C 180,E1 -21860.444,E2 -21860.444} C_VEL
LIN {X 0,Y 191.061,Z 282.729,A -85,B 0,C 180,E1 -21863.665,E2 -21863.665} C_VEL
LIN {X 0,Y 191.896,Z 278.103,A -85,B 0,C 180,E1 -21866.852,E2 -21866.852} C_VEL
LIN {X 0,Y 193.251,Z 271.116,A -85,B 0,C 180,E1 -21870.522,E2 -21870.522} C_VEL
LIN {X 0,Y 194.931,Z 263.554,A -85,B 0,C 180,E1 -21873.618,E2 -21873.618} C_VEL
LIN {X 0,Y 196.716,Z 255.822,A -85,B 0,C 180,E1 -21876.154,E2 -21876.154} C_VEL
LIN {X 0,Y 198.864,Z 245.811,A -85,B 0,C 180,E1 -21878.781,E2 -21878.781} C_VEL
LIN {X 0,Y 201.114,Z 234.632,A -85,B 0,C 180,E1 -21881.082,E2 -21881.082} C_VEL
LIN {X 0,Y 202.748,Z 224.349,A -85,B 0,C 180,E1 -21882.767,E2 -21882.767} C_VEL
LIN {X 0,Y 204.451,Z 212.038,A -85,B 0,C 180,E1 -21884.305,E2 -21884.305} C_VEL
LIN {X 0,Y 205.853,Z 199.077,A -85,B 0,C 180,E1 -21885.47,E2 -21885.47} C_VEL
LIN {X 0,Y 206.709,Z 186.592,A -85,B 0,C 180,E1 -21886.224,E2 -21886.224} C_VEL
LIN {X 0,Y 209.234,Z 123.823,A -85,B 0,C 180,E1 -21888.322,E2 -21888.322} C_VEL
LIN {X 0,Y 202.116,Z 107.272,A -85,B 0,C 180,E1 -21890.024,E2 -21890.024} C_VEL
LIN {X 0,Y 193.959,Z 91.779,A -85,B 0,C 180,E1 -21892.018,E2 -21892.018} C_VEL
LIN {X 0,Y 192.789,Z 89.211,A -85,B 0,C 180,E1 -21892.336,E2 -21892.336} C_VEL
LIN {X 0,Y 192.672,Z 88.477,A -85,B 0,C 180,E1 -21892.433,E2 -21892.433} C_VEL
LIN {X 0,Y 192.665,Z 88.477,A -85,B 0,C 180,E1 -21898.309,E2 -21898.309} C_VEL
LIN {X 0,Y 192.602,Z 88.478,A -85,B 0,C 180,E1 -21903.186,E2 -21903.186} C_VEL
LIN {X 0,Y 192.614,Z 88.49,A -85,B 0,C 180,E1 -21906.608,E2 -21906.608} C_VEL
LIN {X 0,Y 192.552,Z 88.496,A -85,B 0,C 180,E1 -21911.071,E2 -21911.071} C_VEL
LIN {X 0,Y 192.526,Z 88.498,A -85,B 0,C 180,E1 -21916.085,E2 -21916.085} C_VEL
LIN {X 0,Y 192.522,Z 88.496,A -85,B 0,C 180,E1 -21920.051,E2 -21920.051} C_VEL
LIN {X 0,Y 192.563,Z 88.454,A -85,B 0,C 180,E1 -21924.27,E2 -21924.27} C_VEL
LIN {X 0,Y 192.611,Z 88.467,A -85,B 0,C 180,E1 -21927.059,E2 -21927.059} C_VEL
LIN {X 0,Y 192.664,Z 88.485,A -85,B 0,C 180,E1 -21931.691,E2 -21931.691} C_VEL
LIN {X 0,Y 192.71,Z 88.468,A -85,B 0,C 180,E1 -21936.348,E2 -21936.348} C_VEL
LIN {X 0,Y 192.736,Z 88.473,A -85,B 0,C 180,E1 -21941.457,E2 -21941.457} C_VEL
LIN {X 0,Y 192.768,Z 88.466,A -85,B 0,C 180,E1 -21945.213,E2 -21945.213} C_VEL
LIN {X 0,Y 192.948,Z 88.448,A -85,B 0,C 180,E1 -21949.566,E2 -21949.566} C_VEL
LIN {X 0,Y 192.988,Z 88.438,A -85,B 0,C 180,E1 -21953.727,E2 -21953.727} C_VEL
LIN {X 0,Y 193.266,Z 88.406,A -85,B 0,C 180,E1 -21957.916,E2 -21957.916} C_VEL
LIN {X 0,Y 193.446,Z 88.376,A -85,B 0,C 180,E1 -21960,E2 -21960} C_VEL
LIN {X 0,Y 192.974,Z 88.447,A -85,B 0,C 180,E1 -21964.177,E2 -21964.177} C_VEL
LIN {X 0,Y 193.037,Z 88.428,A -85,B 0,C 180,E1 -21968.373,E2 -21968.373} C_VEL
LIN {X 0,Y 192.804,Z 88.468,A -85,B 0,C 180,E1 -21972.633,E2 -21972.633} C_VEL
LIN {X 0,Y 192.76,Z 88.468,A -85,B 0,C 180,E1 -21976.958,E2 -21976.958} C_VEL
LIN {X 0,Y 192.624,Z 88.488,A -85,B 0,C 180,E1 -21981.398,E2 -21981.398} C_VEL
LIN {X 0,Y 192.65,Z 88.486,A -85,B 0,C 180,E1 -21984.213,E2 -21984.213} C_VEL
LIN {X 0,Y 192.652,Z 88.48,A -85,B 0,C 180,E1 -21988.891,E2 -21988.891} C_VEL
LIN {X 0,Y 192.601,Z 88.493,A -85,B 0,C 180,E1 -21993.185,E2 -21993.185} C_VEL
LIN {X 0,Y 192.553,Z 88.501,A -85,B 0,C 180,E1 -21998.351,E2 -21998.351} C_VEL
LIN {X 0,Y 192.493,Z 88.502,A -85,B 0,C 180,E1 -22003.095,E2 -22003.095} C_VEL
LIN {X 0,Y 192.515,Z 88.505,A -85,B 0,C 180,E1 -22006.896,E2 -22006.896} C_VEL
LIN {X 0,Y 192.579,Z 88.609,A -85,B 0,C 180,E1 -22009.068,E2 -22009.068} C_VEL
LIN {X 0,Y 194.416,Z 95.854,A -85,B 0,C 180,E1 -22012.682,E2 -22012.682} C_VEL
LIN {X 0,Y 194.865,Z 97.934,A -85,B 0,C 180,E1 -22013.637,E2 -22013.637} C_VEL
LIN {X 0,Y 202.499,Z 117.024,A -85,B 0,C 180,E1 -22015.661,E2 -22015.661} C_VEL
LIN {X 0,Y 204.381,Z 122.597,A -85,B 0,C 180,E1 -22016.167,E2 -22016.167} C_VEL
LIN {X 0,Y 207.717,Z 156.561,A -85,B 0,C 180,E1 -22017.957,E2 -22017.957} C_VEL
LIN {X 0,Y 207.874,Z 160.399,A -85,B 0,C 180,E1 -22018.125,E2 -22018.125} C_VEL
LIN {X 0,Y 206.837,Z 166.185,A -85,B 0,C 180,E1 -22018.206,E2 -22018.206} C_VEL
LIN {X 0,Y 201.558,Z 181.394,A -85,B 0,C 180,E1 -22018.077,E2 -22018.077} C_VEL
LIN {X 0,Y 200.557,Z 187.322,A -85,B 0,C 180,E1 -22018.173,E2 -22018.173} C_VEL
LIN {X 0,Y 199.551,Z 209.102,A -85,B 0,C 180,E1 -22018.997,E2 -22018.997} C_VEL
LIN {X 0,Y 198.283,Z 221.637,A -85,B 0,C 180,E1 -22019.809,E2 -22019.809} C_VEL
LIN {X 0,Y 196.659,Z 233.988,A -85,B 0,C 180,E1 -22021.007,E2 -22021.007} C_VEL
LIN {X 0,Y 194.602,Z 245.858,A -85,B 0,C 180,E1 -22022.582,E2 -22022.582} C_VEL
LIN {X 0,Y 192.639,Z 256.005,A -85,B 0,C 180,E1 -22024.326,E2 -22024.326} C_VEL
LIN {X 0,Y 190.553,Z 265.469,A -85,B 0,C 180,E1 -22026.353,E2 -22026.353} C_VEL
LIN {X 0,Y 188.541,Z 274.409,A -85,B 0,C 180,E1 -22028.731,E2 -22028.731} C_VEL
LIN {X 0,Y 186.84,Z 282.382,A -85,B 0,C 180,E1 -22031.353,E2 -22031.353} C_VEL
LIN {X 0,Y 185.189,Z 290.293,A -85,B 0,C 180,E1 -22034.594,E2 -22034.594} C_VEL
LIN {X 0,Y 184.022,Z 296.599,A -85,B 0,C 180,E1 -22037.874,E2 -22037.874} C_VEL
LIN {X 0,Y 183.498,Z 301.61,A -85,B 0,C 180,E1 -22041.187,E2 -22041.187} C_VEL
LIN {X 0,Y 183.395,Z 306.046,A -85,B 0,C 180,E1 -22045.108,E2 -22045.108} C_VEL
LIN {X 0,Y 183.453,Z 308.227,A -85,B 0,C 180,E1 -22047.804,E2 -22047.804} C_VEL
LIN {X 0,Y 183.571,Z 309.515,A -85,B 0,C 180,E1 -22049.999,E2 -22049.999} C_VEL
LIN {X 0,Y 183.418,Z 310.376,A -85,B 0,C 180,E1 -22052.195,E2 -22052.195} C_VEL
LIN {X 0,Y 183.323,Z 310.841,A -85,B 0,C 180,E1 -22054.619,E2 -22054.619} C_VEL
LIN {X 0,Y 183.457,Z 310.492,A -85,B 0,C 180,E1 -22058.814,E2 -22058.814} C_VEL
LIN {X 0,Y 184.512,Z 308.643,A -85,B 0,C 180,E1 -22063.21,E2 -22063.21} C_VEL
LIN {X 0,Y 185.421,Z 307.095,A -85,B 0,C 180,E1 -22065.385,E2 -22065.385} C_VEL
LIN {X 0,Y 187.497,Z 304.017,A -85,B 0,C 180,E1 -22068.578,E2 -22068.578} C_VEL
LIN {X 0,Y 190.779,Z 298.69,A -85,B 0,C 180,E1 -22072.469,E2 -22072.469} C_VEL
LIN {X 0,Y 194.192,Z 292.649,A -85,B 0,C 180,E1 -22075.739,E2 -22075.739} C_VEL
LIN {X 0,Y 198.111,Z 285.66,A -85,B 0,C 180,E1 -22078.614,E2 -22078.614} C_VEL
LIN {X 0,Y 202.636,Z 276.945,A -85,B 0,C 180,E1 -22081.348,E2 -22081.348} C_VEL
LIN {X 0,Y 206.734,Z 268.063,A -85,B 0,C 180,E1 -22083.533,E2 -22083.533} C_VEL
LIN {X 0,Y 210.266,Z 259.505,A -85,B 0,C 180,E1 -22085.209,E2 -22085.209} C_VEL
LIN {X 0,Y 214.026,Z 249.128,A -85,B 0,C 180,E1 -22086.817,E2 -22086.817} C_VEL
LIN {X 0,Y 217.549,Z 237.746,A -85,B 0,C 180,E1 -22088.158,E2 -22088.158} C_VEL
LIN {X 0,Y 220.72,Z 224.735,A -85,B 0,C 180,E1 -22089.259,E2 -22089.259} C_VEL
LIN {X 0,Y 222.866,Z 211.742,A -85,B 0,C 180,E1 -22090.053,E2 -22090.053} C_VEL
LIN {X 0,Y 224.136,Z 198.657,A -85,B 0,C 180,E1 -22090.551,E2 -22090.551} C_VEL
LIN {X 0,Y 225.957,Z 168.307,A -85,B 0,C 180,E1 -22091.46,E2 -22091.46} C_VEL
LIN {X 0,Y 224.763,Z 158.436,A -85,B 0,C 180,E1 -22092.249,E2 -22092.249} C_VEL
LIN {X 0,Y 220.47,Z 148.304,A -85,B 0,C 180,E1 -22093.989,E2 -22093.989} C_VEL
LIN {X 0,Y 216.299,Z 139.34,A -85,B 0,C 180,E1 -22095.772,E2 -22095.772} C_VEL
LIN {X 0,Y 212.15,Z 131.473,A -85,B 0,C 180,E1 -22097.636,E2 -22097.636} C_VEL
LIN {X 0,Y 206.996,Z 122.461,A -85,B 0,C 180,E1 -22100.14,E2 -22100.14} C_VEL
LIN {X 0,Y 204.206,Z 117.792,A -85,B 0,C 180,E1 -22101.616,E2 -22101.616} C_VEL
LIN {X 0,Y 200.435,Z 111.929,A -85,B 0,C 180,E1 -22103.751,E2 -22103.751} C_VEL
LIN {X 0,Y 196.454,Z 105.953,A -85,B 0,C 180,E1 -22106.254,E2 -22106.254} C_VEL
LIN {X 0,Y 192.835,Z 101.067,A -85,B 0,C 180,E1 -22108.788,E2 -22108.788} C_VEL
LIN {X 0,Y 191.85,Z 99.496,A -85,B 0,C 180,E1 -22109.561,E2 -22109.561} C_VEL
LIN {X 0,Y 187.236,Z 93.541,A -85,B 0,C 180,E1 -22113.53,E2 -22113.53} C_VEL
LIN {X 0,Y 186.595,Z 92.257,A -85,B 0,C 180,E1 -22114.334,E2 -22114.334} C_VEL
LIN {X 0,Y 185.588,Z 89.355,A -85,B 0,C 180,E1 -22118.624,E2 -22118.624} C_VEL
LIN {X 0,Y 185.688,Z 89.337,A -85,B 0,C 180,E1 -22122.375,E2 -22122.375} C_VEL
LIN {X 0,Y 185.732,Z 89.331,A -85,B 0,C 180,E1 -22126.878,E2 -22126.878} C_VEL
LIN {X 0,Y 186.007,Z 89.301,A -85,B 0,C 180,E1 -22131.308,E2 -22131.308} C_VEL
LIN {X 0,Y 186.206,Z 89.271,A -85,B 0,C 180,E1 -22137.837,E2 -22137.837} C_VEL
LIN {X 0,Y 186.405,Z 89.265,A -85,B 0,C 180,E1 -22140,E2 -22140} C_VEL
LIN {X 0,Y 185.915,Z 89.315,A -85,B 0,C 180,E1 -22144.336,E2 -22144.336} C_VEL
LIN {X 0,Y 185.979,Z 89.302,A -85,B 0,C 180,E1 -22148.695,E2 -22148.695} C_VEL
LIN {X 0,Y 185.802,Z 89.348,A -85,B 0,C 180,E1 -22151.524,E2 -22151.524} C_VEL
LIN {X 0,Y 186.339,Z 91.401,A -85,B 0,C 180,E1 -22152.249,E2 -22152.249} C_VEL
LIN {X 0,Y 187.984,Z 93.741,A -85,B 0,C 180,E1 -22153.872,E2 -22153.872} C_VEL
LIN {X 0,Y 190.68,Z 95.457,A -85,B 0,C 180,E1 -22156.048,E2 -22156.048} C_VEL
LIN {X 0,Y 192.202,Z 98.321,A -85,B 0,C 180,E1 -22157.339,E2 -22157.339} C_VEL
LIN {X 0,Y 194.701,Z 100.624,A -85,B 0,C 180,E1 -22159.095,E2 -22159.095} C_VEL
LIN {X 0,Y 195.711,Z 102.164,A -85,B 0,C 180,E1 -22159.811,E2 -22159.811} C_VEL
LIN {X 0,Y 198.122,Z 105.201,A -85,B 0,C 180,E1 -22161.373,E2 -22161.373} C_VEL
LIN {X 0,Y 199.382,Z 106.512,A -85,B 0,C 180,E1 -22162.123,E2 -22162.123} C_VEL
LIN {X 0,Y 202.177,Z 110.203,A -85,B 0,C 180,E1 -22163.742,E2 -22163.742} C_VEL
LIN {X 0,Y 203.407,Z 111.858,A -85,B 0,C 180,E1 -22164.42,E2 -22164.42} C_VEL
LIN {X 0,Y 207.127,Z 116.907,A -85,B 0,C 180,E1 -22166.353,E2 -22166.353} C_VEL
LIN {X 0,Y 212.149,Z 124.014,A -85,B 0,C 180,E1 -22168.726,E2 -22168.726} C_VEL
LIN {X 0,Y 218.605,Z 134.053,A -85,B 0,C 180,E1 -22171.487,E2 -22171.487} C_VEL
LIN {X 0,Y 224.77,Z 144.907,A -85,B 0,C 180,E1 -22173.895,E2 -22173.895} C_VEL
LIN {X 0,Y 227.16,Z 149.525,A -85,B 0,C 180,E1 -22174.781,E2 -22174.781} C_VEL
LIN {X 0,Y 224.565,Z 189.067,A -85,B 0,C 180,E1 -22175.977,E2 -22175.977} C_VEL
LIN {X 0,Y 222.802,Z 202.934,A -85,B 0,C 180,E1 -22176.733,E2 -22176.733} C_VEL
LIN {X 0,Y 220.582,Z 215.257,A -85,B 0,C 180,E1 -22177.764,E2 -22177.764} C_VEL
LIN {X 0,Y 217.456,Z 227.503,A -85,B 0,C 180,E1 -22179.136,E2 -22179.136} C_VEL
LIN {X 0,Y 213.801,Z 239.191,A -85,B 0,C 180,E1 -22180.884,E2 -22180.884} C_VEL
LIN {X 0,Y 209.824,Z 249.553,A -85,B 0,C 180,E1 -22182.888,E2 -22182.888} C_VEL
LIN {X 0,Y 206.071,Z 257.998,A -85,B 0,C 180,E1 -22184.955,E2 -22184.955} C_VEL
LIN {X 0,Y 202.16,Z 265.837,A -85,B 0,C 180,E1 -22187.371,E2 -22187.371} C_VEL
LIN {X 0,Y 198.09,Z 273.257,A -85,B 0,C 180,E1 -22190.312,E2 -22190.312} C_VEL
LIN {X 0,Y 194.453,Z 279.207,A -85,B 0,C 180,E1 -22193.392,E2 -22193.392} C_VEL
LIN {X 0,Y 191.27,Z 283.804,A -85,B 0,C 180,E1 -22196.555,E2 -22196.555} C_VEL
